// TIA Portal V16 program export: 8 tag tables, 6 data types, 67 data blocks, 106 code blocks (in call order from the OBs), 61 instance data blocks

VAR_GLOBAL   // PLC tag table "Default tag table"
   START AT %M0.0 : Bool;
   OUTPUT AT %M0.2 : Bool;
   STOP AT %M0.1 : Bool;
   MW100 AT %MW100 : Int;
END_VAR

VAR_GLOBAL   // PLC tag table "Analógicas"
   FQ301_MEDIDOR_CAUDAL AT %IW16 : Word;
   PC401_SENSOR_PRESSÃO AT %IW18 : Word;
END_VAR

VAR_GLOBAL   // PLC tag table "Estados_Componentes"
   BS001A_ON AT %I1.5 : Bool;
   BS001A_DISPARO AT %I2.0 : Bool;
   BS001B_ON AT %I2.1 : Bool;
   BS001B_DISPARO AT %I2.2 : Bool;
   XV102_ABERTA AT %I2.3 : Bool;
   XV102_FECHADA AT %I2.4 : Bool;
   XV101_ABERTA AT %I2.5 : Bool;
   MX201_ON AT %I2.6 : Bool;
   MX201_DISPARO AT %I2.7 : Bool;
   BH201_ON AT %I3.0 : Bool;
   BH201_DISPARO AT %I3.1 : Bool;
   MX301_ON AT %I3.2 : Bool;
   MX301_DISPARO AT %I3.3 : Bool;
   BM401_ON AT %I3.4 : Bool;
   BM401_DISPARO AT %I3.5 : Bool;
   BS501_ON AT %I3.6 : Bool;
   BS501_DISPARO AT %I3.7 : Bool;
   MX601_ON AT %I4.0 : Bool;
   MX601_DISPARO AT %I4.1 : Bool;
   BD601_ON AT %I4.2 : Bool;
   BD601_DISPARO AT %I4.3 : Bool;
   BD602_ON AT %I4.4 : Bool;
   BD602_DISPARO AT %I4.5 : Bool;
   MX603_ON AT %I4.6 : Bool;
   MX603_DISPARO AT %I4.7 : Bool;
   BD603_ON AT %I5.0 : Bool;
   BD603_DISPARO AT %I5.1 : Bool;
   MX604_ON AT %I5.2 : Bool;
   MX604_DISPARO AT %I5.3 : Bool;
   BD604_ON AT %I5.4 : Bool;
   BD604_DISPARO AT %I5.5 : Bool;
   MX605_ON AT %I5.6 : Bool;
   MX605_DISPARO AT %I5.7 : Bool;
   BD605_ON AT %I6.0 : Bool;
   BD605_DISPARO AT %I6.1 : Bool;
   BOT_EMERGÊNCIA AT %I6.2 : Bool;
   PH201_CONT_PH AT %I6.3 : Bool;
   PH301_CONT_PH AT %I6.4 : Bool;
   TEMPERATURA_ATINGIDA AT %I6.5 : Bool;
   RH201_CONT_REDOX AT %I6.6 : Bool;
END_VAR

VAR_GLOBAL   // PLC tag table "Falhas"
   DISPARO_DIF_3Q1_32 AT %I0.0 : Bool;
   DISPARO_DIFERENCIAL_3Q3 AT %I0.1 : Bool;
   DISPARO_DIFERENCIAL_4Q1_4Q2 AT %I0.2 : Bool;
   FALHA_24VDC AT %I0.3 : Bool;
   FALHA_220VAC AT %I0.4 : Bool;
   FALHA_24VAC AT %I0.5 : Bool;
END_VAR

VAR_GLOBAL   // PLC tag table "Níveis"
   LSH001_TK00 AT %I0.6 : Bool;
   LSL001_TK00 AT %I1.0 : Bool;
   LSH501_TK05 AT %I1.3 : Bool;
   LSL501_TK05 AT %I1.4 : Bool;
   LSH101_TK01 AT %I1.1 : Bool;
   LS201_TK02 AT %IW12 : Word;
   LS301_TK03 AT %IW14 : Word;
   LSL101_TK01 AT %I1.2 : Bool;
   LSM001_TK00 AT %I0.7 : Bool;
END_VAR

VAR_GLOBAL   // PLC tag table "Saídas"
   BS001A AT %Q0.0 : Bool;
   BS001B AT %Q0.1 : Bool;
   XV101 AT %Q3.3 : Bool;
   XV102 AT %Q3.4 : Bool;
   MX201 AT %Q0.4 : Bool;
   BH201 AT %Q0.5 : Bool;
   MX301 AT %Q0.6 : Bool;
   ALIM_BM401 AT %Q0.7 : Bool;
   LIGAR_BM401 AT %Q3.1 : Bool;
   BS501 AT %Q1.1 : Bool;
   MX601 AT %Q2.0 : Bool;
   BD601 AT %Q2.1 : Bool;
   BD602 AT %Q2.2 : Bool;
   MX603 AT %Q2.3 : Bool;
   BD603 AT %Q2.4 : Bool;
   MX604 AT %Q2.5 : Bool;
   BD604 AT %Q2.6 : Bool;
   MX605 AT %Q2.7 : Bool;
   BD605 AT %Q0.2 : Bool;
   ALARME AT %Q3.2 : Bool;
END_VAR

VAR_GLOBAL   // PLC tag table "Inputs"
   "EV1.1_ABERTA" AT %I0.0 : Bool;
   "EV1.1_FECHADA" AT %I0.1 : Bool;
   "EV2.1_ABERTA" AT %I0.2 : Bool;
   "EV2.1_FECHADA" AT %I0.3 : Bool;
   "EV3.1_ABERTA" AT %I0.4 : Bool;
   "EV3.1_FECHADA" AT %I0.5 : Bool;
   "EV4.1_ABERTA" AT %I0.6 : Bool;
   "EV4.1_FECHADA" AT %I0.7 : Bool;
   "EV5.1_ABERTA" AT %I1.0 : Bool;
   "EV5.1_FECHADA" AT %I1.1 : Bool;
   "EV1.2_ABERTA" AT %I1.2 : Bool;
   "EV1.2_FECHADA" AT %I1.3 : Bool;
   "EV2.2_ABERTA" AT %I1.4 : Bool;
   "EV2.2_FECHADA" AT %I1.5 : Bool;
   "EV3.2_ABERTA" AT %I2.0 : Bool;
   "EV3.2_FECHADA" AT %I2.1 : Bool;
   "EV4.2_ABERTA" AT %I2.2 : Bool;
   "EV4.2_FECHADA" AT %I2.3 : Bool;
   "EV5.2_ABERTA" AT %I2.4 : Bool;
   "EV5.2_FECHADA" AT %I2.5 : Bool;
   PRESSOSTATO_1 AT %IW4 : Word;
   PRESSOSTATO_2 AT %IW6 : Word;
   AVARIA_BOMBA_1 AT %I2.6 : Bool;
   AVARIA_BOMBA_2 AT %I2.7 : Bool;
   AVARIA_BOMBA_3 AT %I3.0 : Bool;
END_VAR

VAR_GLOBAL   // PLC tag table "Outputs"
   "EV1.1" AT %Q0.0 : Bool;
   "EV2.1" AT %Q0.1 : Bool;
   "EV3.1" AT %Q0.2 : Bool;
   "EV4.1" AT %Q0.3 : Bool;
   "EV5.1" AT %Q0.4 : Bool;
   "EV1.2" AT %Q0.5 : Bool;
   "EV2.2" AT %Q0.6 : Bool;
   "EV3.2" AT %Q0.7 : Bool;
   "EV4.2" AT %Q1.0 : Bool;
   "EV5.2" AT %Q1.1 : Bool;
   BOMBA_1_VAR AT %Q2.0 : Bool;
   BOMBA_2_VAR AT %Q2.1 : Bool;
   BOMBA_3_RESERVA AT %Q2.2 : Bool;
   ULTRAVIOLETA AT %Q2.3 : Bool;
END_VAR

TYPE "InverterData"
// stored: IsFailsafeCompliant false
   STRUCT
      control_word : Word;
      setpoint : Real;
      ref_quantity : Struct
         speed_p2000 : Real;
         current_p2002 : Real;
         torque_p2003 : Real;
      END_STRUCT;
      status_word : Word;
      actual_speed : Real;
      actual_current : Real;
      actual_torque : Real;
      actual_alarm : Word;
      actual_fault : Word;
      RETVAL_RD : Word;
      RETVAL_WR : Word;
   END_STRUCT;
END_TYPE

TYPE "APP"
// stored: IsFailsafeCompliant false
   STRUCT
      PID_ComponenteProporzionale : DInt;
      PID_ComponenteIntegrale : DInt;
      PID_ComponenteDerivativa : DInt;
      Tiro : Int;   // Valore di tiro richiesto: 1-100 => 1-100% Setup 1, 101-200 => 1-100% Setup 2, 0 => Azzera regolatore
      Tiro1 : Int;
      Tiro2 : Int;
      TiroPrecedente : Int;   // Valore di tiro richiesto istante (n-1)
      TiroAppoggio : Int;
      ErroreAttuale : Int;   // Errore istante (n)
      ErrorePrecedente : Int;   // Errore istante (n-1)
      PID_Kp : Int;   // Kp in uso nel PID
      PID_Ki : Int;   // Ki in uso nel PID
      PID_Kd : Int;   // Kd in uso nel PID
      SetpointTiro : Int;   // Valore di setpoint del PID
      SetpointTiroRampa : Int;   // Valore di setpoint del PID iniziale a rampa
      TransitorioInizialeFase1 : Int;   // Indica che si deve eseguire la rampa iniziale (Fase 1)
      TransitorioFase3 : Int;   // Indica che si deve eseguire la rampa da velocita' alta a media (Fase 3)
      TransitorioFase4 : Int;   // Indica che si deve eseguire la rampa da velocita' media a bassa (Fase 4)
      VelocitaRotazione : Int;   // Velocita' di rotazione richiesta
      VelocitaRotazioneFase2 : Int;   // Velocita' di rotazione richiesta durante la Fase 2
      VelocitaRotazioneAppoggio1 : Int;
      VelocitaRotazioneAppoggio2 : Int;
      Fase1OneShoot : Int;   // Indica che sono appena entrato nella fase di traansitorio di accelerazione (Fase 1)
      Fase2OneShoot : Int;   // Indica che sono appena entrato nella fase di transitorio iniziale (Fase 2)
      Fase3OneShoot : Int;   // Indica che sono appena entrato nella fase di transitorio di velocita' alta - media (Fase 3)
      Fase4OneShoot : Int;   // Indica che sono appena entrato nella fase di transitorio di velocita' media - bassa (Fase 4)
      ArrestoRepentinoOneShoot : Int;   // Indica che sono appena entrato nella fase di arresto repentino
      TiroFase1 : Int;   // Indica il tiro nella Fase 1 usato nella Fase 2
      TempIntero : Int;
      Fase : Int;
      BallerinoPrecedente : Array[0..2] of Int;   // Valore del ballerino negli istanti precedenti
      LimiteComponenteIntegrale : Int;   // Limite della componente integrale durante la transizione dalla velocita alta a media (Fase 3) e dalla media a bassa (Fase 4)
      TiroRichiesto : Int;   // Valore di tiro compreso fra 1 e 100 richiesto dalla logica di controllo
      TimerArrestoRepentino : Int;   // Timer per arresto repentino.
      TiroMinimoArrestoRepentino : Int;   // Tiro minimo durante un'arresto repentino
      VariazioneTiro : Int;   // Variazione del tiro film (ballerino)
      TimerFase2 : Int;   // Timer usato nella Fase 2 per arrestare i rulli in caso di rottura film
      TempoRotturaFilm : Int;   // Tempo rottura film in numero di scansioni (1 scansione ogni 30msec)
      TimerFase4 : Int;   // Timer per Fase 4
      TiroMinimoFase4 : Int;   // Tiro minimo durante la Fase 4 di arresto
      PID_Uscita : DInt;   // Valore di uscita del PID
      PrestiroRichiesto : DInt;   // Valore di prestiro richiesto. Valore compreso fra 0 e 500
      PrestiroAppoggio : Real;
   END_STRUCT;
END_TYPE

TYPE "DatiProgramma"
// stored: IsFailsafeCompliant false
   STRUCT
      Wrapping : Bool;   // Wrapping (0=Excluded 1=Included)
      TopLenght : Int;   // Top film lenght
      TopRelease : Int;   // Top carriage release position
      TopDown : Int;   // Top carriage downward to release top film
      Top : Int;   // Top cycle (1=Excluded 2=Before 3=Waterp-2 4=Waterp-3 5=Waterp-4)
      PressurePTime : Int;   // Time for pressure plate downward
      LifterTime : Int;   // Time for pallet lifter upward
      RevOverContrast : Int;   // Revolution over welder contrast
      RopeEndCycle : Byte;   // Rope type at end of cycle (Program)
      Spare4 : Byte;
      RopeTime : Int;   // Delay for rope unit opened
      RevOverClamp : Int;   // Revolution over clamp
      FilmForceFinalRev : Int;   // Film force on the final revolutions
      FilmPrestretchFinalRev : Int;   // Film prestretch on the final revolutions
      ArmSpeed : Int;   // Arm rotation speed (%*10)
      CarriageDown4Top : Int;   // Spool carriage downward for top cycle
      TopDownTime : Int;   // Top carriage downward for top cycle
      LapsUnderTop : Int;   // Revolutions under top film
      Spare6 : Int;   // Spare
      Spare7 : Int;   // Spare
      Spare8 : Int;   // Spare
      Spare9 : Int;   // Spare
      Spare10 : Int;   // Spare
      Spare11 : Int;   // Spare
      Spare12 : Int;   // Spare
      Overlap0_1 : Int := 0;   // Film overlap spool carriage height 0->1
      Height1 : Int := 0;   // Spool carriage height 1 (mm)
      Landmark1 : Bool := false;   // Landmark for spool carriage height 1 (0=Bottom 1=Top)
      Lifter1 : Bool := false;   // Pallet lifter for spool carriage height 1
      SpareBit1H1 : Bool := false;   // Spare bit for spool carriage height 1 (Program)
      Airblower1 : Bool := false;   // Airblower on film tail for spool carriage height 1 (0=Excluded 1=Included)
      NextStep1 : Bool := false;   // Next step for spool carriage height 1 (0=End 1=Next)
      PressureP1 : Bool := false;   // Pressure plate for spool carriage height 1 (0=Excluded 1=Included)
      SpareByte2H1 : Byte := 16#0;   // Spare byte for spool carriage height 1
      Revolution1 : Int := 0;   // Revolutions for spool carriage height 1
      RopeUnit1_1 : Byte := 16#0;   // Rope unit for spool carriage height 1 (1=Excluded 2=Inc 3=Inc during)
      RopeUnit1_2 : Byte := 16#0;   // Rope unit for spool carriage height 1 (1=Excluded 2=Inc 3=Inc during)
      FilmForce1 : Int := 0;   // Film force for spool carriage height 1
      FilmPrestretch1 : Int := 0;   // Film prestretch for spool carriage height 1
      Spare3H1 : Int := 0;   // Spare for spool carriage height 1
      Spare49 : Int := 0;   // Spare
      Spare50 : Int := 0;   // Spare
      Spare51 : Int := 0;   // Spare
      Spare52 : Int := 0;   // Spare
      Spare53 : Int := 0;   // Spare
      Overlap1_2 : Int := 0;   // Film overlap spool carriage height 1->2
      Height2 : Int := 0;   // Spool carriage height 2 (mm)
      Landmark2 : Bool := false;   // Landmark for spool carriage height 2 (0=Bottom 1=Top)
      Lifter2 : Bool := false;   // Pallet lifter for spool carriage height 2
      SpareBit1H2 : Bool := false;   // Spare bit for spool carriage height 2
      Airblower2 : Bool := false;   // Airblower on film tail for spool carriage height 2 (0=Excluded 1=Included)
      NextStep2 : Bool := false;   // Next step for spool carriage height 2 (0=End 1=Next)
      PressureP2 : Bool := false;   // Pressure plate for spool carriage height 2 (0=Excluded 1=Included)
      SpareByte2H2 : Byte := 16#0;   // Spare byte for spool carriage height 2
      Revolution2 : Int := 0;   // Revolutions for spool carriage height 2
      RopeUnit2_1 : Byte := 16#0;   // Rope unit for spool carriage height 2 (1=Excluded 2=Inc 3=Inc during)
      RopeUnit2_2 : Byte := 16#0;   // Rope unit for spool carriage height 2 (1=Excluded 2=Inc 3=Inc during)
      FilmForce2 : Int := 0;   // Film force for spool carriage height 2
      FilmPrestretch2 : Int := 0;   // Film prestretch for spool carriage height 2
      Spare3H2 : Int := 0;   // Spare for spool carriage height 2
      Spare54 : Int := 0;   // Spare
      Spare55 : Int := 0;   // Spare
      Spare56 : Int := 0;   // Spare
      Spare57 : Int := 0;   // Spare
      Spare58 : Int := 0;   // Spare
      Overlap2_3 : Int := 0;   // Film overlap spool carriage height 2->3
      Height3 : Int := 0;   // Spool carriage height 3 (mm)
      Landmark3 : Bool := false;   // Landmark for spool carriage height 3 (0=Bottom 1=Top)
      Lifter3 : Bool := false;   // Pallet lifter for spool carriage height 3
      SpareBit1H3 : Bool := false;   // Spare bit for spool carriage height 3
      Airblower3 : Bool := false;   // Airblower on film tail for spool carriage height 3 (0=Excluded 1=Included)
      NextStep3 : Bool := false;   // Next step for spool carriage height 3 (0=End 1=Next)
      PressureP3 : Bool := false;   // Pressure plate for spool carriage height 3 (0=Excluded 1=Included)
      SpareByte2H3 : Byte := 16#0;   // Spare byte for spool carriage height 3
      Revolution3 : Int := 0;   // Revolutions for spool carriage height 3
      RopeUnit3_1 : Byte := 16#0;   // Rope unit for spool carriage height 3 (1=Excluded 2=Inc 3=Inc during)
      RopeUnit3_2 : Byte := 16#0;   // Rope unit for spool carriage height 3 (1=Excluded 2=Inc 3=Inc during)
      FilmForce3 : Int := 0;   // Film force for spool carriage height 3
      FilmPrestretch3 : Int := 0;   // Film prestretch for spool carriage height 3
      Spare3H3 : Int := 0;   // Spare for spool carriage height 3
      Spare59 : Int := 0;   // Spare
      Spare60 : Int := 0;   // Spare
      Spare61 : Int := 0;   // Spare
      Spare62 : Int := 0;   // Spare
      Spare63 : Int := 0;   // Spare
      Overlap3_4 : Int := 0;   // Film overlap spool carriage height 3->4
      Height4 : Int := 0;   // Spool carriage height 4 (mm)
      Landmark4 : Bool := false;   // Landmark for spool carriage height 4 (0=Bottom 1=Top)
      Lifter4 : Bool := false;   // Pallet lifter for spool carriage height 4
      SpareBit1H4 : Bool := false;   // Spare bit for spool carriage height 4
      Airblower4 : Bool := false;   // Airblower on film tail for spool carriage height 4 (0=Excluded 1=Included)
      NextStep4 : Bool := false;   // Next step for spool carriage height 4 (0=End 1=Next)
      PressureP4 : Bool := false;   // Pressure plate for spool carriage height 4 (0=Excluded 1=Included)
      SpareByte2H4 : Byte := 16#0;   // Spare byte for spool carriage height 4
      Revolution4 : Int := 0;   // Revolutions for spool carriage height 4
      RopeUnit4_1 : Byte := 16#0;   // Rope unit for spool carriage height 4 (1=Excluded 2=Inc 3=Inc during)
      RopeUnit4_2 : Byte := 16#0;   // Rope unit for spool carriage height 4 (1=Excluded 2=Inc 3=Inc during)
      FilmForce4 : Int := 0;   // Film force for spool carriage height 4
      FilmPrestretch4 : Int := 0;   // Film prestretch for spool carriage height 4
      Spare3H4 : Int := 0;   // Spare for spool carriage height 4
      Spare64 : Int := 0;   // Spare
      Spare65 : Int := 0;   // Spare
      Spare66 : Int := 0;   // Spare
      Spare67 : Int := 0;   // Spare
      Spare68 : Int := 0;   // Spare
      Overlap4_5 : Int := 0;   // Film overlap spool carriage height 4->5
      Height5 : Int := 0;   // Spool carriage height 5 (mm)
      Landmark5 : Bool := false;   // Landmark for spool carriage height 5 (0=Bottom 1=Top)
      Lifter5 : Bool := false;   // Pallet lifter for spool carriage height 5
      SpareBit1H5 : Bool := false;   // Spare bit for spool carriage height 5
      Airblower5 : Bool := false;   // Airblower on film tail for spool carriage height 5 (0=Excluded 1=Included)
      NextStep5 : Bool := false;   // Next step for spool carriage height 5 (0=End 1=Next)
      PressureP5 : Bool := false;   // Pressure plate for spool carriage height 5 (0=Excluded 1=Included)
      SpareByte2H5 : Byte := 16#0;   // Spare byte for spool carriage height 5
      Revolution5 : Int := 0;   // Revolutions for spool carriage height 5
      RopeUnit5_1 : Byte := 16#0;   // Rope unit for spool carriage height 5 (1=Excluded 2=Inc 3=Inc during)
      RopeUnit5_2 : Byte := 16#0;   // Rope unit for spool carriage height 5 (1=Excluded 2=Inc 3=Inc during)
      FilmForce5 : Int := 0;   // Film force for spool carriage height 5
      FilmPrestretch5 : Int := 0;   // Film prestretch for spool carriage height 5
      Spare3H5 : Int := 0;   // Spare for spool carriage height 5
      Spare69 : Int := 0;   // Spare
      Spare70 : Int := 0;   // Spare
      Spare71 : Int := 0;   // Spare
      Spare72 : Int := 0;   // Spare
      Spare73 : Int := 0;   // Spare
      Overlap5_6 : Int := 0;   // Film overlap spool carriage height 5->6
      Height6 : Int := 0;   // Spool carriage height 6 (mm)
      Landmark6 : Bool := false;   // Landmark for spool carriage height 6 (0=Bottom 1=Top)
      Lifter6 : Bool := false;   // Pallet lifter for spool carriage height 6
      SpareBit1H6 : Bool := false;   // Spare bit for spool carriage height 6
      Airblower6 : Bool := false;   // Airblower on film tail for spool carriage height 6 (0=Excluded 1=Included)
      NextStep6 : Bool := false;   // Next step for spool carriage height 6 (0=End 1=Next)
      PressureP6 : Bool := false;   // Pressure plate for spool carriage height 6 (0=Excluded 1=Included)
      SpareByte2H6 : Byte := 16#0;   // Spare byte for spool carriage height 6
      Revolution6 : Int := 0;   // Revolutions for spool carriage height 6
      RopeUnit6_1 : Byte := 16#0;   // Rope unit for spool carriage height 6 (1=Excluded 2=Inc 3=Inc during)
      RopeUnit6_2 : Byte := 16#0;   // Rope unit for spool carriage height 6 (1=Excluded 2=Inc 3=Inc during)
      FilmForce6 : Int := 0;   // Film force for spool carriage height 6
      FilmPrestretch6 : Int := 0;   // Film prestretch for spool carriage height 6
      Spare3H6 : Int := 0;   // Spare for spool carriage height 6
      Spare74 : Int := 0;   // Spare
      Spare75 : Int := 0;   // Spare
      Spare76 : Int := 0;   // Spare
      Spare77 : Int := 0;   // Spare
      Spare78 : Int := 0;   // Spare
      Overlap6_7 : Int := 0;   // Film overlap spool carriage height 6->7
      Height7 : Int := 0;   // Spool carriage height 7 (mm)
      Landmark7 : Bool := false;   // Landmark for spool carriage height 7 (0=Bottom 1=Top)
      Lifter7 : Bool := false;   // Pallet lifter for spool carriage height 7
      SpareBit1H7 : Bool := false;   // Spare bit for spool carriage height 7
      Airblower7 : Bool := false;   // Airblower on film tail for spool carriage height 7 (0=Excluded 1=Included)
      NextStep7 : Bool := false;   // Next step for spool carriage height 7 (0=End 1=Next)
      PressureP7 : Bool := false;   // Pressure plate for spool carriage height 7 (0=Excluded 1=Included)
      SpareByte2H7 : Byte := 16#0;   // Spare byte for spool carriage height 7
      Revolution7 : Int := 0;   // Revolutions for spool carriage height 7
      RopeUnit7_1 : Byte := 16#0;   // Rope unit for spool carriage height 7 (1=Excluded 2=Inc 3=Inc during)
      RopeUnit7_2 : Byte := 16#0;   // Rope unit for spool carriage height 7 (1=Excluded 2=Inc 3=Inc during)
      FilmForce7 : Int := 0;   // Film force for spool carriage height 7
      FilmPrestretch7 : Int := 0;   // Film prestretch for spool carriage height 7
      Spare3H7 : Int := 0;   // Spare for spool carriage height 7
      Spare79 : Int := 0;   // Spare
      Spare80 : Int := 0;   // Spare
      Spare81 : Int := 0;   // Spare
      Spare82 : Int := 0;   // Spare
      Spare83 : Int := 0;   // Spare
      Overlap7_8 : Int := 0;   // Film overlap spool carriage height 7->8
      Height8 : Int := 0;   // Spool carriage height 8 (mm)
      Landmark8 : Bool := false;   // Landmark for spool carriage height 8 (0=Bottom 1=Top)
      Lifter8 : Bool := false;   // Pallet lifter for spool carriage height 8
      SpareBit1H8 : Bool := false;   // Spare bit for spool carriage height 8
      Airblower8 : Bool := false;   // Airblower on film tail for spool carriage height 8 (0=Excluded 1=Included)
      NextStep8 : Bool := false;   // Next step for spool carriage height 8 (0=End 1=Next)
      PressureP8 : Bool := false;   // Pressure plate for spool carriage height 8 (0=Excluded 1=Included)
      SpareByte2H8 : Byte := 16#0;   // Spare byte for spool carriage height 8
      Revolution8 : Int := 0;   // Revolutions for spool carriage height 8
      RopeUnit8_1 : Byte := 16#0;   // Rope unit for spool carriage height 8 (1=Excluded 2=Inc 3=Inc during)
      RopeUnit8_2 : Byte := 16#0;   // Rope unit for spool carriage height 8 (1=Excluded 2=Inc 3=Inc during)
      FilmForce8 : Int := 0;   // Film force for spool carriage height 8
      FilmPrestretch8 : Int := 0;   // Film prestretch for spool carriage height 8
      Spare3H8 : Int := 0;   // Spare for spool carriage height 8
      Spare84 : Int := 0;   // Spare
      Spare85 : Int := 0;   // Spare
      Spare86 : Int := 0;   // Spare
      Spare87 : Int := 0;   // Spare
      Spare88 : Int := 0;   // Spare
      Overlap8_9 : Int := 0;   // Film overlap spool carriage height 8->9
      Height9 : Int := 0;   // Spool carriage height 9 (mm)
      Landmark9 : Bool := false;   // Landmark for spool carriage height 9 (0=Bottom 1=Top)
      Lifter9 : Bool := false;   // Pallet lifter for spool carriage height 9
      SpareBit1H9 : Bool := false;   // Spare bit for spool carriage height 9
      Airblower9 : Bool := false;   // Airblower on film tail for spool carriage height 9 (0=Excluded 1=Included)
      NextStep9 : Bool := false;   // Next step for spool carriage height 9 (0=End 1=Next)
      PressureP9 : Bool := false;   // Pressure plate for spool carriage height 9 (0=Excluded 1=Included)
      SpareByte2H9 : Byte := 16#0;   // Spare byte for spool carriage height 9
      Revolution9 : Int := 0;   // Revolutions for spool carriage height 9
      RopeUnit9_1 : Byte := 16#0;   // Rope unit for spool carriage height 9 (1=Excluded 2=Inc 3=Inc during)
      RopeUnit9_2 : Byte := 16#0;   // Rope unit for spool carriage height 9 (1=Excluded 2=Inc 3=Inc during)
      FilmForce9 : Int := 0;   // Film force for spool carriage height 9
      FilmPrestretch9 : Int := 0;   // Film prestretch for spool carriage height 9
      Spare3H9 : Int := 0;   // Spare for spool carriage height 9
      Spare89 : Int := 0;   // Spare
      Spare90 : Int := 0;   // Spare
      Spare91 : Int := 0;   // Spare
      Spare92 : Int := 0;   // Spare
      Spare93 : Int := 0;   // Spare
      Overlap9_10 : Int := 0;   // Film overlap spool carriage height 9->10
      Height10 : Int := 0;   // Spool carriage height 10 (mm)
      Landmark10 : Bool := false;   // Landmark for spool carriage height 10 (0=Bottom 1=Top)
      Lifter10 : Bool := false;   // Pallet lifter for spool carriage height 10
      SpareBit1H10 : Bool := false;   // Spare bit for spool carriage height 10
      Airblower10 : Bool := false;   // Airblower on film tail for spool carriage height 10 (0=Excluded 1=Included)
      NextStep10 : Bool := false;   // Next step for spool carriage height 10 (0=End 1=Next)
      PressureP10 : Bool := false;   // Pressure plate for spool carriage height 10 (0=Excluded 1=Included)
      SpareByte2H10 : Byte := 16#0;   // Spare byte for spool carriage height 10
      Revolution10 : Int := 0;   // Revolutions for spool carriage height 10
      RopeUnit10_1 : Byte := 16#0;   // Rope unit for spool carriage height 10 (1=Excluded 2=Inc 3=Inc during)
      RopeUnit10_2 : Byte := 16#0;   // Rope unit for spool carriage height 10 (1=Excluded 2=Inc 3=Inc during)
      FilmForce10 : Int := 0;   // Film force for spool carriage height 10
      FilmPrestretch10 : Int := 0;   // Film prestretch for spool carriage height 10
      Spare3H10 : Int := 0;   // Spare for spool carriage height 10
      Spare94 : Int := 0;   // Spare
      Spare95 : Int := 0;   // Spare
      Spare96 : Int := 0;   // Spare
      Spare97 : Int := 0;   // Spare
      Spare98 : Int := 0;   // Spare
      Overlap10_11 : Int := 0;   // Film overlap spool carriage height 10->11
      Height11 : Int := 0;   // Spool carriage height 11 (mm)
      Landmark11 : Bool := false;   // Landmark for spool carriage height 11 (0=Bottom 1=Top)
      Lifter11 : Bool := false;   // Pallet lifter for spool carriage height 11
      SpareBit1H11 : Bool := false;   // Spare bit for spool carriage height 11
      Airblower11 : Bool := false;   // Airblower on film tail for spool carriage height 11 (0=Excluded 1=Included)
      NextStep11 : Bool := false;   // Next step for spool carriage height 11 (0=End 1=Next)
      PressureP11 : Bool := false;   // Pressure plate for spool carriage height 11 (0=Excluded 1=Included)
      SpareByte2H11 : Byte := 16#0;   // Spare byte for spool carriage height 11
      Revolution11 : Int := 0;   // Revolutions for spool carriage height 11
      RopeUnit11_1 : Byte := 16#0;   // Rope unit for spool carriage height 11 (1=Excluded 2=Inc 3=Inc during)
      RopeUnit11_2 : Byte := 16#0;   // Rope unit for spool carriage height 11 (1=Excluded 2=Inc 3=Inc during)
      FilmForce11 : Int := 0;   // Film force for spool carriage height 11
      FilmPrestretch11 : Int := 0;   // Film prestretch for spool carriage height 11
      Spare3H11 : Int := 0;   // Spare for spool carriage height 11
      Spare99 : Int := 0;   // Spare
      Spare100 : Int := 0;   // Spare
      Spare101 : Int := 0;   // Spare
      Spare102 : Int := 0;   // Spare
      Spare103 : Int := 0;   // Spare
      Overlap11_12 : Int := 0;   // Film overlap spool carriage height 11->12
      Height12 : Int := 0;   // Spool carriage height 12 (mm)
      Landmark12 : Bool := false;   // Landmark for spool carriage height 12 (0=Bottom 1=Top)
      Lifter12 : Bool := false;   // Pallet lifter for spool carriage height 12
      SpareBit1H12 : Bool := false;   // Spare bit for spool carriage height 12
      Airblower12 : Bool := false;   // Airblower on film tail for spool carriage height 12 (0=Excluded 1=Included)
      NextStep12 : Bool := false;   // Next step for spool carriage height 12 (0=End 1=Next)
      PressureP12 : Bool := false;   // Pressure plate for spool carriage height 12 (0=Excluded 1=Included)
      SpareByte2H12 : Byte := 16#0;   // Spare byte for spool carriage height 12
      Revolution12 : Int := 0;   // Revolutions for spool carriage height 12
      RopeUnit12_1 : Byte := 16#0;   // Rope unit for spool carriage height 12 (1=Excluded 2=Inc 3=Inc during)
      RopeUnit12_2 : Byte := 16#0;   // Rope unit for spool carriage height 12 (1=Excluded 2=Inc 3=Inc during)
      FilmForce12 : Int := 0;   // Film force for spool carriage height 12
      FilmPrestretch12 : Int := 0;   // Film prestretch for spool carriage height 12
      Spare3H12 : Int := 0;   // Spare for spool carriage height 12
      Spare104 : Int := 0;   // Spare
      Spare105 : Int := 0;   // Spare
      Spare106 : Int := 0;   // Spare
      Spare107 : Int := 0;   // Spare
      Spare108 : Int := 0;   // Spare
   END_STRUCT;
END_TYPE

TYPE "M20"
// stored: IsFailsafeCompliant false
   STRUCT
      M20_P00 : Int;   // Tipo di prestiro
      M20_P01 : Int;   // Coefficiente proporzionale per il regolatore PID
      M20_P02 : Int;   // Coefficiente integrale (Fase1 e Fase2) per il regolatore PID
      M20_P03 : Int;   // Coefficiente derivativo per il regolatore PID
      M20_P04 : Int;   // Coefficiente integrale (Fase3 e Fase4) per il regolatore PID
      M20_P05 : Int;   // Rampa di accelerazione per il tiro durante la Fase1
      M20_P06 : Int;   // Limite componente integrale nel transitorio dalla Fase2 alla Fase3
      M20_P07 : Int;   // Limite componente integrale nel transitorio dalla Fase3 alla Fase4
      M20_P08 : Int;   // Valore minimo ingresso analogico
      M20_P09 : Int;   // Valore massimo ingresso analogico
      M20_P10 : Int;   // Prestiro naturale dovuto al rapporto di riduzione
      M20_P11 : Int;   // Velocità per il jog in manuale dei rulli di prestiro
      M20_P12 : Int;   // Offset del rullo lento 10 equivale a 0
      M20_P13 : Int;   // Jog di velocità durante la partenza del braccio
      M20_P14 : Int;   // Tiro minimo durante la Fase4 di arresto e durante un arresto repentino
      M20_P15 : Int;   // Tempo (in decimi di secondo) dopo il quale i rulli si fermano per rottura film
      M20_P20 : Int;   // Velocità indicata da plc per la rotazione braccio e il carrello top
      M20_P21 : Int;   // Velocità indicata da plc per il carrello di prestiro e il trasporto di centro macchina
      M20_P22 : Int;   // Tiro indicato da plc
      M20_P23 : Int;   // Prestiro indicato da plc
      M20_P24 : Int;   // Valore di ingresso analogico AI0
      M20_P25 : Int;   // Tiro richiesto da plc compreso fra 0 e 100
   END_STRUCT;
END_TYPE

TYPE "PID"
// stored: IsFailsafeCompliant false
   STRUCT
      proporzionale : DInt;
      integrativo : DInt;
      segnale : DInt;
      maxSegnale : Int;
      minSegnale : Int;
      setPointShow : UInt;
      tiro : UInt;
      vParP : UInt;
      vParI : UInt;
      svuota : Bool;
      attiva : Bool;
      setTiro : Bool;
      "timer" : Time;
   END_STRUCT;
END_TYPE

TYPE "ProgramDataGreyBar"
// stored: IsFailsafeCompliant false
   STRUCT
      Overlap : Int;   // Film overlap
      Height : Int;   // Spool carriage height (mm)
      Landmark : Bool;   // Landmark (0=Bottom 1=Top)
      Lifter : Bool;   // Pallet lifter
      SpareBit1 : Bool;   // Spare
      Airblower : Bool;   // Airblower on film tail (0=Excluded 1=Included)
      NextStep : Bool;   // Next step (0=End 1=Next)
      PressureP : Bool;   // Pressure plate (0=Excluded 1=Included)
      SpareByte1 : Byte;   // Spare
      Revolution : Int;   // Revolutions
      RopeUnitUpper : Byte;   // Upper rope unit (1=Exc 2=Inc 3=Inc during)
      RopeUnitLower : Byte;   // Lower rope unit (1=Exc 2=Inc 3=Inc during)
      FilmForce : Int;   // Film force
      FilmPrestretch : Int;   // Film prestretch
      SpareWord1 : Int;   // Spare
      SpareWord2 : Int;   // Spare
      SpareWord3 : Int;   // Spare
      SpareWord4 : Int;   // Spare
      SpareWord5 : Int;   // Spare
      SpareWord6 : Int;   // Spare
   END_STRUCT;
END_TYPE

DATA_BLOCK "Data_block_1"   // DB1
{ S7_Optimized_Access := 'TRUE' }
VERSION : 0.1
// stored: AutoNumber true, DBAccessibleFromOPCUA true, IsOnlyStoredInLoadMemory false, IsRetainMemResEnabled false, IsWriteProtectedInAS false, MemoryReserve 100
   VAR
      DADOS : Byte;
   END_VAR
BEGIN
END_DATA_BLOCK

DATA_BLOCK "DB04_Conveyor"   // DB4
{ S7_Optimized_Access := 'FALSE' }
AUTHOR : Robopac
VERSION : 0.0
// stored: AutoNumber false, IsOnlyStoredInLoadMemory false, IsWriteProtectedInAS false
   VAR RETAIN
      dbw0 : Int := 0;
      dbw2 : Int := 0;
      dbx4_0 : Bool := TRUE;   // Pallet positioned
      dbx4_1 : Bool := FALSE;   // Deceleration for pallet positioning
      dbx4_2 : Bool := FALSE;   // Support memory for wrong pallet positioning emergency
      dbx4_3 : Bool := FALSE;   // Unload memory for outfeed conveyor
      dbx4_4 : Bool := TRUE;   // Support for end of transfer signal for pallet load/unload
      dbx4_5 : Bool := TRUE;   // Short pallet positioned
      dbx4_6 : Bool := TRUE;   // Pallet positioned for clampcutcycle
      dbx4_7 : Bool := FALSE;   // Pallet positioned from reverse
      dbb5 : Byte := 16#00;
      dbw6 : Int := 0;
      dbw8 : Int := 0;
      dbw10 : Int := 0;   // Pallet lenght measured in infeed (pulse)
      dbw12 : Int := 0;   // Pallet lenght measured in central machine (pulse)
      dbw14 : Int := 0;   // Pallet lenght measured in infeed (mm)
      dbw16 : Int := 0;   // Pallet lenght measured in central machine (mm)
      dbw18 : Int := 0;   // Half pallet lenght for selfcentering system
      dbw20 : Int := -100;   // Deceleration for pallet positioning on selfcentering system
      dbw22 : Int := 78;   // Support for conveyor movement speed
      dbw24 : Int := 0;
      dbw26 : Int := 0;
      dbw28 : Int := 0;
      dbw30 : Int := 0;
      dbw32 : Int := 0;
      dbw34 : Int := 0;
      dbd36 : DInt := 0;
      dbd40 : DInt := 0;
      dbd44 : DInt := 0;
      dbd48 : DInt := 0;
      dbd52 : DInt := 0;
      dbd56 : DInt := 0;
      dbd60 : DInt := 0;
      dbd64 : DInt := 0;
      dbd68 : DInt := 0;
      dbd72 : DInt := 0;
      dbw76 : Int := 0;
      dbb78 : Byte := 16#00;   // Rope unit for running spool carriage height (1=Excluded 2=Inc 3=Inc during
      dbb79 : Byte := 16#00;   // Rope unit for running spool carriage height (1=Excluded 2=Inc 3=Inc during
      dbd80 : DInt := 0;
      dbd84 : DInt := 0;
   END_VAR
BEGIN
END_DATA_BLOCK

DATA_BLOCK "DB09_TablePos"   // DB9
{ S7_Optimized_Access := 'FALSE' }
AUTHOR : Robopac
VERSION : 0.0
// stored: AutoNumber false, IsOnlyStoredInLoadMemory false, IsWriteProtectedInAS false
   VAR RETAIN
      dbx0_0 : Bool := FALSE;
      dbx0_1 : Bool := FALSE;
      dbx0_2 : Bool := TRUE;
      dbx0_3 : Bool := FALSE;
      dbx0_4 : Bool := FALSE;
      dbx0_5 : Bool := FALSE;
      dbx0_6 : Bool := FALSE;
      dbx0_7 : Bool := FALSE;
      dbx1_0 : Bool := FALSE;   // Table rotation axis movement forward
      dbx1_1 : Bool := FALSE;   // Table rotation axis movement backward
      dbx1_2 : Bool := FALSE;   // Table rotation axis movement inside low speed area
      dbx1_3 : Bool := FALSE;   // Table rotation axis movement low speed
      dbx1_4 : Bool := FALSE;   // Table rotation forward
      dbx1_5 : Bool := FALSE;   // Table rotation backward
      dbx1_6 : Bool := TRUE;
      dbx1_7 : Bool := FALSE;
      dbx2_0 : Bool := FALSE;
      dbx2_1 : Bool := FALSE;
      dbx2_2 : Bool := FALSE;
      dbx2_3 : Bool := FALSE;
      dbx2_4 : Bool := FALSE;
      dbx2_5 : Bool := FALSE;
      dbx2_6 : Bool := FALSE;
      dbx2_7 : Bool := FALSE;
      dbx3_0 : Bool := FALSE;   // Table rotation: Support for encoder running control
      dbx3_1 : Bool := FALSE;   // Table rotation: Support for encoder running control alarm
      dbx3_2 : Bool := FALSE;
      dbx3_3 : Bool := FALSE;
      dbx3_4 : Bool := FALSE;
      dbx3_5 : Bool := FALSE;
      dbx3_6 : Bool := FALSE;
      dbx3_7 : Bool := FALSE;
      dbx4_0 : Bool := FALSE;
      dbx4_1 : Bool := FALSE;
      dbx4_2 : Bool := FALSE;
      dbx4_3 : Bool := FALSE;
      dbx4_4 : Bool := FALSE;
      dbx4_5 : Bool := FALSE;
      dbx4_6 : Bool := FALSE;
      dbx4_7 : Bool := FALSE;
      dbx5_0 : Bool := FALSE;
      dbx5_1 : Bool := FALSE;
      dbx5_2 : Bool := FALSE;
      dbx5_3 : Bool := FALSE;
      dbw6 : Int := 5;   // Table rotation: Support for movement speed
      dbw8 : Int := 0;   // Table rotation: Support for movement deceleration
      dbw10 : Int := 5;   // Table rotation inverter: Support for speed selection
      dbw12 : Int := 10199;
      dbw14 : Int := 2340;
      dbw16 : Int := 0;
      dbw18 : Int := 0;
      dbw20 : Int := 0;
      dbw22 : Int := 0;
      dbw24 : Int := 0;
      dbw26 : Int := 0;
      dbw28 : Int := 0;
      dbd30 : DInt := -15;   // Table rotation position: Pulse
      dbw34 : Int := -8;   // Table position
      dbw36 : Int := 0;   // Table rotation position: Table maximum position
      dbw38 : Int := 0;   // Table rotation position: Deceleration position
      dbw40 : Int := 0;   // Table rotation position: Deceleration position
      dbd42 : DInt := -15;   // Support for encoder table rotation running control
      dbw46 : Int := 20;   // Support for encoder table rotation running control
      dbw48 : Int := -8;   // Table position according to offset
      dbw50 : Int := 0;
      dbw52 : Int := 0;
      dbw54 : Int := 0;
      dbw56 : Int := 0;
      dbw58 : Int := 0;
      dbw60 : Int := 0;
      dbw62 : Int := 0;
      dbw64 : Int := 0;
      dbw66 : Int := 0;
      dbw68 : Int := 0;
      dbw70 : Int := 0;
      Req1_Dest : Int := 0;   // Positioning request 1: Destination position
      Req2_Dest : Int := 0;   // Positioning request 2: Destination position
      Req3_Dest : Int := 0;   // Positioning request 3: Destination position
      Req4_Dest : Int := 0;   // Positioning request 4: Destination position
      Req1_Fwd : Bool := FALSE;   // Positioning request 1: Axis forward
      Req1_Bkw : Bool := FALSE;   // Positioning request 1: Axis backward
      Req1_Slow : Bool := FALSE;   // Positioning request 1: Axis slow speed
      Req1_Pos : Bool := FALSE;   // Positioning request 1: Axis in position
      Req2_Fwd : Bool := FALSE;   // Positioning request 2: Axis forward
      Req2_Bkw : Bool := FALSE;   // Positioning request 2: Axis backward
      Req2_Slow : Bool := FALSE;   // Positioning request 2: Axis slow speed
      Req2_Pos : Bool := FALSE;   // Positioning request 2: Axis in position
      Req3_Fwd : Bool := FALSE;   // Positioning request 3: Axis forward
      Req3_Bkw : Bool := FALSE;   // Positioning request 3: Axis backward
      Req3_Slow : Bool := FALSE;   // Positioning request 3: Axis slow speed
      Req3_Pos : Bool := FALSE;   // Positioning request 3: Axis in position
      Req4_Fwd : Bool := FALSE;   // Positioning request 4: Axis forward
      Req4_Bkw : Bool := FALSE;   // Positioning request 4: Axis backward
      Req4_Slow : Bool := FALSE;   // Positioning request 4: Axis slow speed
      Req4_Pos : Bool := FALSE;   // Positioning request 4: Axis in position
      Req5_Dest : Int := 0;   // Positioning request 4: Destination position
      Req6_Dest : Int := 0;   // Positioning request 4: Destination position
      Req7_Dest : Int := 0;   // Positioning request 4: Destination position
      Req8_Dest : Int := 0;   // Positioning request 4: Destination position
      Req5_Fwd : Bool := FALSE;   // Positioning request 5: Axis forward
      Req5_Bkw : Bool := FALSE;   // Positioning request 5: Axis backward
      Req5_Slow : Bool := FALSE;   // Positioning request 5: Axis slow speed
      Req5_Pos : Bool := FALSE;   // Positioning request 5: Axis in position
      Req6_Fwd : Bool := FALSE;   // Positioning request 6: Axis forward
      Req6_Bkw : Bool := FALSE;   // Positioning request 6: Axis backward
      Req6_Slow : Bool := FALSE;   // Positioning request 6: Axis slow speed
      Req6_Pos : Bool := FALSE;   // Positioning request 6: Axis in position
      Req7_Fwd : Bool := FALSE;   // Positioning request 7: Axis forward
      Req7_Bkw : Bool := FALSE;   // Positioning request 7: Axis backward
      Req7_Slow : Bool := FALSE;   // Positioning request 7: Axis slow speed
      Req7_Pos : Bool := FALSE;   // Positioning request 7: Axis in position
      Req8_Fwd : Bool := FALSE;   // Positioning request 8: Axis forward
      Req8_Bkw : Bool := FALSE;   // Positioning request 8: Axis backward
      Req8_Slow : Bool := FALSE;   // Positioning request 8: Axis slow speed
      Req8_Pos : Bool := FALSE;   // Positioning request 8: Axis in position
      dbw92 : Int := 0;
      dbw94 : Int := 0;
      dbw96 : Int := 0;
      dbw98 : Int := 0;
   END_VAR
BEGIN
END_DATA_BLOCK

DATA_BLOCK "DB13_TableFaseControl"   // DB13
{ S7_Optimized_Access := 'FALSE' }
VERSION : 0.1
// stored: AutoNumber false, IsOnlyStoredInLoadMemory false, IsWriteProtectedInAS false
   VAR RETAIN
      load : Bool := TRUE;
      cm : Bool := TRUE;
      unload : Bool := TRUE;
      hysteresis : Int := 100;
   END_VAR
BEGIN
END_DATA_BLOCK

DATA_BLOCK "DB18_TableSpeed"   // DB18
{ S7_Optimized_Access := 'FALSE' }
VERSION : 0.1
// stored: AutoNumber false, IsOnlyStoredInLoadMemory false, IsWriteProtectedInAS false
   VAR RETAIN
      spare0 : Int := 0;
      spare1 : Int := 0;
      spare2 : Int := 0;
      spare3 : Int := 0;
      spare4 : Int := 0;
      spare5 : Int := 0;
      spare6 : Int := 0;
      spare7 : Int := 0;
      DBD16 : Real := 0.0;   // Actual speed in degrees per second (split before use)
      DBD20 : Real := 90.0;   // Low speed in degrees per second (split before use)
      DBD24 : Real := 900.0;   // High speed in degrees per second (split before use)
      spare14 : Int := 0;
      DBW30 : Int := 0;   // Degrees to reach minimum speed from maximum speed
      spare16 : Int := 0;
      DBW34 : Int := 50;
   END_VAR
BEGIN
END_DATA_BLOCK

DATA_BLOCK "DB21_DisplayGeneralData"   // DB21
{ S7_Optimized_Access := 'FALSE' }
AUTHOR : Robopac
VERSION : 0.0
// stored: AutoNumber false, IsOnlyStoredInLoadMemory false, IsWriteProtectedInAS false
   VAR RETAIN
      dbx0_0 : Bool := TRUE;   // Welder unit included(1)/excluded (Display-General Data)
      dbx0_1 : Bool := FALSE;   // Machine included(1)/excluded (Display-General Data)
      dbx0_2 : Bool := TRUE;   // Pallet load/unload included(1)/excluded (Display-Sysdata)
      dbx0_3 : Bool := TRUE;   // Load pallet with forklift selection by display (Display-Sysdata)
      dbx0_4 : Bool := TRUE;   // Unload pallet with forklift selection by display (Display-Sysdata)
      dbx0_5 : Bool := FALSE;
      dbx0_6 : Bool := TRUE;
      dbx0_7 : Bool := FALSE;
      dbb1 : Byte := 16#00;
      dbw2 : Int := 3;   // PLC SW major release
      dbw4 : Int := 0;   // PLC SW minor release
      dbw6 : Int := 90;   // Spool carriage upward for spring clamp at begin cycle (Display-General Data)
      dbw8 : Int := 0;   // Spool carriage downward for film tail at the cycle begin (Display-General Data)
      dbw10 : Int := 2;   // Film thickness (Display-General Data)
      dbw12 : Int := 700;   // Welding time (Display-General Data)
      dbw14 : Int := 0;   // Low speed for Helix conveyor movement (%) (Display-Sysdata)
      dbw16 : Int := 0;   // High speed for Helix conveyor movement (%) (Display-Sysdata)
      dbw18 : Int := 500;   // Delay on pallet positioning (Display-General Data)
      dbw20 : Int := 10000;   // Delay for load/unload pallet simultaneously (Display-General Data)
      dbw22 : Int := 100;   // Deceleration for pallet positioning (Display-General Data)
      dbw24 : Int := 1;   // Time for pallet load with forklift
      dbw26 : Int := 0;   // Override for ring movement in manul mode (Display-General Data)
      dbw28 : Int := 100;   // TIMER CICLO FIERA (attesa tra cicli successivi)
      dbw30 : Int := 0;   // Film prestretch for film prestretch test cycle (Display-General Data)
      dbw32 : Int := 0;   // Film prestretch increase for film prestretch test (Display-General Data)
      dbw34 : Int := 0;   // Film supplied every revolution for film prestretch test (Display-General Data)
      dbw36 : Int := 0;   // Time for spool carriage upward for table cycle (Display-Sysdata)
      dbw38 : Int := 2000;   // Time for spool carriage upward for table cycle (Display-Sysdata)
      dbw40 : Int := 15000;   // Time load with forklift
      dbw42 : Int := 10000;   // Time unload with forklift
   END_VAR
BEGIN
END_DATA_BLOCK

DATA_BLOCK "DB234_Program16"   // DB234
{ S7_Optimized_Access := 'FALSE' }
AUTHOR : Robopac
VERSION : 0.0
// stored: AutoNumber false, IsOnlyStoredInLoadMemory false, IsWriteProtectedInAS false
   VAR RETAIN
      Program16 { S7_SetPoint := 'True'} : "DatiProgramma";
   END_VAR
BEGIN
   Program16.Wrapping := FALSE;
   Program16.TopLenght := 0;
   Program16.TopRelease := 0;
   Program16.TopDown := 0;
   Program16.Top := 0;
   Program16.PressurePTime := 0;
   Program16.LifterTime := 0;
   Program16.RevOverContrast := 0;
   Program16.RopeEndCycle := 16#00;
   Program16.Spare4 := 16#00;
   Program16.RopeTime := 0;
   Program16.RevOverClamp := 0;
   Program16.FilmForceFinalRev := 0;
   Program16.FilmPrestretchFinalRev := 0;
   Program16.ArmSpeed := 0;
   Program16.CarriageDown4Top := 0;
   Program16.TopDownTime := 0;
   Program16.LapsUnderTop := 0;
   Program16.Spare6 := 0;
   Program16.Spare7 := 0;
   Program16.Spare8 := 0;
   Program16.Spare9 := 0;
   Program16.Spare10 := 0;
   Program16.Spare11 := 0;
   Program16.Spare12 := 0;
   Program16.Overlap0_1 := 0;
   Program16.Height1 := 0;
   Program16.Landmark1 := FALSE;
   Program16.Lifter1 := FALSE;
   Program16.SpareBit1H1 := FALSE;
   Program16.Airblower1 := FALSE;
   Program16.NextStep1 := FALSE;
   Program16.PressureP1 := FALSE;
   Program16.SpareByte2H1 := 16#00;
   Program16.Revolution1 := 0;
   Program16.RopeUnit1_1 := 16#00;
   Program16.RopeUnit1_2 := 16#00;
   Program16.FilmForce1 := 0;
   Program16.FilmPrestretch1 := 0;
   Program16.Spare3H1 := 0;
   Program16.Spare49 := 0;
   Program16.Spare50 := 0;
   Program16.Spare51 := 0;
   Program16.Spare52 := 0;
   Program16.Spare53 := 0;
   Program16.Overlap1_2 := 0;
   Program16.Height2 := 0;
   Program16.Landmark2 := FALSE;
   Program16.Lifter2 := FALSE;
   Program16.SpareBit1H2 := FALSE;
   Program16.Airblower2 := FALSE;
   Program16.NextStep2 := FALSE;
   Program16.PressureP2 := FALSE;
   Program16.SpareByte2H2 := 16#00;
   Program16.Revolution2 := 0;
   Program16.RopeUnit2_1 := 16#00;
   Program16.RopeUnit2_2 := 16#00;
   Program16.FilmForce2 := 0;
   Program16.FilmPrestretch2 := 0;
   Program16.Spare3H2 := 0;
   Program16.Spare54 := 0;
   Program16.Spare55 := 0;
   Program16.Spare56 := 0;
   Program16.Spare57 := 0;
   Program16.Spare58 := 0;
   Program16.Overlap2_3 := 0;
   Program16.Height3 := 0;
   Program16.Landmark3 := FALSE;
   Program16.Lifter3 := FALSE;
   Program16.SpareBit1H3 := FALSE;
   Program16.Airblower3 := FALSE;
   Program16.NextStep3 := FALSE;
   Program16.PressureP3 := FALSE;
   Program16.SpareByte2H3 := 16#00;
   Program16.Revolution3 := 0;
   Program16.RopeUnit3_1 := 16#00;
   Program16.RopeUnit3_2 := 16#00;
   Program16.FilmForce3 := 0;
   Program16.FilmPrestretch3 := 0;
   Program16.Spare3H3 := 0;
   Program16.Spare59 := 0;
   Program16.Spare60 := 0;
   Program16.Spare61 := 0;
   Program16.Spare62 := 0;
   Program16.Spare63 := 0;
   Program16.Overlap3_4 := 0;
   Program16.Height4 := 0;
   Program16.Landmark4 := FALSE;
   Program16.Lifter4 := FALSE;
   Program16.SpareBit1H4 := FALSE;
   Program16.Airblower4 := FALSE;
   Program16.NextStep4 := FALSE;
   Program16.PressureP4 := FALSE;
   Program16.SpareByte2H4 := 16#00;
   Program16.Revolution4 := 0;
   Program16.RopeUnit4_1 := 16#00;
   Program16.RopeUnit4_2 := 16#00;
   Program16.FilmForce4 := 0;
   Program16.FilmPrestretch4 := 0;
   Program16.Spare3H4 := 0;
   Program16.Spare64 := 0;
   Program16.Spare65 := 0;
   Program16.Spare66 := 0;
   Program16.Spare67 := 0;
   Program16.Spare68 := 0;
   Program16.Overlap4_5 := 0;
   Program16.Height5 := 0;
   Program16.Landmark5 := FALSE;
   Program16.Lifter5 := FALSE;
   Program16.SpareBit1H5 := FALSE;
   Program16.Airblower5 := FALSE;
   Program16.NextStep5 := FALSE;
   Program16.PressureP5 := FALSE;
   Program16.SpareByte2H5 := 16#00;
   Program16.Revolution5 := 0;
   Program16.RopeUnit5_1 := 16#00;
   Program16.RopeUnit5_2 := 16#00;
   Program16.FilmForce5 := 0;
   Program16.FilmPrestretch5 := 0;
   Program16.Spare3H5 := 0;
   Program16.Spare69 := 0;
   Program16.Spare70 := 0;
   Program16.Spare71 := 0;
   Program16.Spare72 := 0;
   Program16.Spare73 := 0;
   Program16.Overlap5_6 := 0;
   Program16.Height6 := 0;
   Program16.Landmark6 := FALSE;
   Program16.Lifter6 := FALSE;
   Program16.SpareBit1H6 := FALSE;
   Program16.Airblower6 := FALSE;
   Program16.NextStep6 := FALSE;
   Program16.PressureP6 := FALSE;
   Program16.SpareByte2H6 := 16#00;
   Program16.Revolution6 := 0;
   Program16.RopeUnit6_1 := 16#00;
   Program16.RopeUnit6_2 := 16#00;
   Program16.FilmForce6 := 0;
   Program16.FilmPrestretch6 := 0;
   Program16.Spare3H6 := 0;
   Program16.Spare74 := 0;
   Program16.Spare75 := 0;
   Program16.Spare76 := 0;
   Program16.Spare77 := 0;
   Program16.Spare78 := 0;
   Program16.Overlap6_7 := 0;
   Program16.Height7 := 0;
   Program16.Landmark7 := FALSE;
   Program16.Lifter7 := FALSE;
   Program16.SpareBit1H7 := FALSE;
   Program16.Airblower7 := FALSE;
   Program16.NextStep7 := FALSE;
   Program16.PressureP7 := FALSE;
   Program16.SpareByte2H7 := 16#00;
   Program16.Revolution7 := 0;
   Program16.RopeUnit7_1 := 16#00;
   Program16.RopeUnit7_2 := 16#00;
   Program16.FilmForce7 := 0;
   Program16.FilmPrestretch7 := 0;
   Program16.Spare3H7 := 0;
   Program16.Spare79 := 0;
   Program16.Spare80 := 0;
   Program16.Spare81 := 0;
   Program16.Spare82 := 0;
   Program16.Spare83 := 0;
   Program16.Overlap7_8 := 0;
   Program16.Height8 := 0;
   Program16.Landmark8 := FALSE;
   Program16.Lifter8 := FALSE;
   Program16.SpareBit1H8 := FALSE;
   Program16.Airblower8 := FALSE;
   Program16.NextStep8 := FALSE;
   Program16.PressureP8 := FALSE;
   Program16.SpareByte2H8 := 16#00;
   Program16.Revolution8 := 0;
   Program16.RopeUnit8_1 := 16#00;
   Program16.RopeUnit8_2 := 16#00;
   Program16.FilmForce8 := 0;
   Program16.FilmPrestretch8 := 0;
   Program16.Spare3H8 := 0;
   Program16.Spare84 := 0;
   Program16.Spare85 := 0;
   Program16.Spare86 := 0;
   Program16.Spare87 := 0;
   Program16.Spare88 := 0;
   Program16.Overlap8_9 := 0;
   Program16.Height9 := 0;
   Program16.Landmark9 := FALSE;
   Program16.Lifter9 := FALSE;
   Program16.SpareBit1H9 := FALSE;
   Program16.Airblower9 := FALSE;
   Program16.NextStep9 := FALSE;
   Program16.PressureP9 := FALSE;
   Program16.SpareByte2H9 := 16#00;
   Program16.Revolution9 := 0;
   Program16.RopeUnit9_1 := 16#00;
   Program16.RopeUnit9_2 := 16#00;
   Program16.FilmForce9 := 0;
   Program16.FilmPrestretch9 := 0;
   Program16.Spare3H9 := 0;
   Program16.Spare89 := 0;
   Program16.Spare90 := 0;
   Program16.Spare91 := 0;
   Program16.Spare92 := 0;
   Program16.Spare93 := 0;
   Program16.Overlap9_10 := 0;
   Program16.Height10 := 0;
   Program16.Landmark10 := FALSE;
   Program16.Lifter10 := FALSE;
   Program16.SpareBit1H10 := FALSE;
   Program16.Airblower10 := FALSE;
   Program16.NextStep10 := FALSE;
   Program16.PressureP10 := FALSE;
   Program16.SpareByte2H10 := 16#00;
   Program16.Revolution10 := 0;
   Program16.RopeUnit10_1 := 16#00;
   Program16.RopeUnit10_2 := 16#00;
   Program16.FilmForce10 := 0;
   Program16.FilmPrestretch10 := 0;
   Program16.Spare3H10 := 0;
   Program16.Spare94 := 0;
   Program16.Spare95 := 0;
   Program16.Spare96 := 0;
   Program16.Spare97 := 0;
   Program16.Spare98 := 0;
   Program16.Overlap10_11 := 0;
   Program16.Height11 := 0;
   Program16.Landmark11 := FALSE;
   Program16.Lifter11 := FALSE;
   Program16.SpareBit1H11 := FALSE;
   Program16.Airblower11 := FALSE;
   Program16.NextStep11 := FALSE;
   Program16.PressureP11 := FALSE;
   Program16.SpareByte2H11 := 16#00;
   Program16.Revolution11 := 0;
   Program16.RopeUnit11_1 := 16#00;
   Program16.RopeUnit11_2 := 16#00;
   Program16.FilmForce11 := 0;
   Program16.FilmPrestretch11 := 0;
   Program16.Spare3H11 := 0;
   Program16.Spare99 := 0;
   Program16.Spare100 := 0;
   Program16.Spare101 := 0;
   Program16.Spare102 := 0;
   Program16.Spare103 := 0;
   Program16.Overlap11_12 := 0;
   Program16.Height12 := 0;
   Program16.Landmark12 := FALSE;
   Program16.Lifter12 := FALSE;
   Program16.SpareBit1H12 := FALSE;
   Program16.Airblower12 := FALSE;
   Program16.NextStep12 := FALSE;
   Program16.PressureP12 := FALSE;
   Program16.SpareByte2H12 := 16#00;
   Program16.Revolution12 := 0;
   Program16.RopeUnit12_1 := 16#00;
   Program16.RopeUnit12_2 := 16#00;
   Program16.FilmForce12 := 0;
   Program16.FilmPrestretch12 := 0;
   Program16.Spare3H12 := 0;
   Program16.Spare104 := 0;
   Program16.Spare105 := 0;
   Program16.Spare106 := 0;
   Program16.Spare107 := 0;
   Program16.Spare108 := 0;
END_DATA_BLOCK

DATA_BLOCK "DB236_Program14"   // DB236
{ S7_Optimized_Access := 'FALSE' }
AUTHOR : Robopac
VERSION : 0.0
// stored: AutoNumber false, IsOnlyStoredInLoadMemory false, IsWriteProtectedInAS false
   VAR RETAIN
      Program14 { S7_SetPoint := 'True'} : "DatiProgramma";
   END_VAR
BEGIN
   Program14.Wrapping := TRUE;
   Program14.TopLenght := 500;
   Program14.TopRelease := 0;
   Program14.TopDown := 0;
   Program14.Top := 4;
   Program14.PressurePTime := 0;
   Program14.LifterTime := 0;
   Program14.RevOverContrast := 1;
   Program14.RopeEndCycle := 16#02;
   Program14.Spare4 := 16#01;
   Program14.RopeTime := 1500;
   Program14.RevOverClamp := 1;
   Program14.FilmForceFinalRev := 10;
   Program14.FilmPrestretchFinalRev := 100;
   Program14.ArmSpeed := 100;
   Program14.CarriageDown4Top := 500;
   Program14.TopDownTime := 1500;
   Program14.LapsUnderTop := 0;
   Program14.Spare6 := 0;
   Program14.Spare7 := 0;
   Program14.Spare8 := 0;
   Program14.Spare9 := 0;
   Program14.Spare10 := 0;
   Program14.Spare11 := 0;
   Program14.Spare12 := 0;
   Program14.Overlap0_1 := 0;
   Program14.Height1 := 130;
   Program14.Landmark1 := FALSE;
   Program14.Lifter1 := FALSE;
   Program14.SpareBit1H1 := FALSE;
   Program14.Airblower1 := TRUE;
   Program14.NextStep1 := TRUE;
   Program14.PressureP1 := TRUE;
   Program14.SpareByte2H1 := 16#00;
   Program14.Revolution1 := 1;
   Program14.RopeUnit1_1 := 16#01;
   Program14.RopeUnit1_2 := 16#01;
   Program14.FilmForce1 := 5;
   Program14.FilmPrestretch1 := 200;
   Program14.Spare3H1 := 0;
   Program14.Spare49 := 0;
   Program14.Spare50 := 0;
   Program14.Spare51 := 0;
   Program14.Spare52 := 0;
   Program14.Spare53 := 0;
   Program14.Overlap1_2 := 0;
   Program14.Height2 := 50;
   Program14.Landmark2 := FALSE;
   Program14.Lifter2 := FALSE;
   Program14.SpareBit1H2 := FALSE;
   Program14.Airblower2 := TRUE;
   Program14.NextStep2 := TRUE;
   Program14.PressureP2 := TRUE;
   Program14.SpareByte2H2 := 16#00;
   Program14.Revolution2 := 1;
   Program14.RopeUnit2_1 := 16#01;
   Program14.RopeUnit2_2 := 16#01;
   Program14.FilmForce2 := 20;
   Program14.FilmPrestretch2 := 200;
   Program14.Spare3H2 := 0;
   Program14.Spare54 := 0;
   Program14.Spare55 := 0;
   Program14.Spare56 := 0;
   Program14.Spare57 := 0;
   Program14.Spare58 := 0;
   Program14.Overlap2_3 := 100;
   Program14.Height3 := -50;
   Program14.Landmark3 := TRUE;
   Program14.Lifter3 := FALSE;
   Program14.SpareBit1H3 := FALSE;
   Program14.Airblower3 := TRUE;
   Program14.NextStep3 := TRUE;
   Program14.PressureP3 := TRUE;
   Program14.SpareByte2H3 := 16#00;
   Program14.Revolution3 := 2;
   Program14.RopeUnit3_1 := 16#01;
   Program14.RopeUnit3_2 := 16#01;
   Program14.FilmForce3 := 30;
   Program14.FilmPrestretch3 := 200;
   Program14.Spare3H3 := 0;
   Program14.Spare59 := 0;
   Program14.Spare60 := 0;
   Program14.Spare61 := 380;
   Program14.Spare62 := 2800;
   Program14.Spare63 := 0;
   Program14.Overlap3_4 := 100;
   Program14.Height4 := 100;
   Program14.Landmark4 := FALSE;
   Program14.Lifter4 := FALSE;
   Program14.SpareBit1H4 := FALSE;
   Program14.Airblower4 := TRUE;
   Program14.NextStep4 := TRUE;
   Program14.PressureP4 := TRUE;
   Program14.SpareByte2H4 := 16#00;
   Program14.Revolution4 := 3;
   Program14.RopeUnit4_1 := 16#02;
   Program14.RopeUnit4_2 := 16#02;
   Program14.FilmForce4 := 30;
   Program14.FilmPrestretch4 := 200;
   Program14.Spare3H4 := 0;
   Program14.Spare64 := 0;
   Program14.Spare65 := 0;
   Program14.Spare66 := 0;
   Program14.Spare67 := 0;
   Program14.Spare68 := 0;
   Program14.Overlap4_5 := 0;
   Program14.Height5 := 50;
   Program14.Landmark5 := FALSE;
   Program14.Lifter5 := FALSE;
   Program14.SpareBit1H5 := FALSE;
   Program14.Airblower5 := TRUE;
   Program14.NextStep5 := FALSE;
   Program14.PressureP5 := FALSE;
   Program14.SpareByte2H5 := 16#00;
   Program14.Revolution5 := 1;
   Program14.RopeUnit5_1 := 16#01;
   Program14.RopeUnit5_2 := 16#01;
   Program14.FilmForce5 := 30;
   Program14.FilmPrestretch5 := 200;
   Program14.Spare3H5 := 0;
   Program14.Spare69 := 0;
   Program14.Spare70 := 0;
   Program14.Spare71 := 0;
   Program14.Spare72 := 0;
   Program14.Spare73 := 0;
   Program14.Overlap5_6 := 100;
   Program14.Height6 := 50;
   Program14.Landmark6 := FALSE;
   Program14.Lifter6 := FALSE;
   Program14.SpareBit1H6 := FALSE;
   Program14.Airblower6 := TRUE;
   Program14.NextStep6 := FALSE;
   Program14.PressureP6 := FALSE;
   Program14.SpareByte2H6 := 16#00;
   Program14.Revolution6 := 2;
   Program14.RopeUnit6_1 := 16#02;
   Program14.RopeUnit6_2 := 16#01;
   Program14.FilmForce6 := 20;
   Program14.FilmPrestretch6 := 200;
   Program14.Spare3H6 := 0;
   Program14.Spare74 := 0;
   Program14.Spare75 := 0;
   Program14.Spare76 := 0;
   Program14.Spare77 := 0;
   Program14.Spare78 := 0;
   Program14.Overlap6_7 := 0;
   Program14.Height7 := 0;
   Program14.Landmark7 := FALSE;
   Program14.Lifter7 := FALSE;
   Program14.SpareBit1H7 := FALSE;
   Program14.Airblower7 := FALSE;
   Program14.NextStep7 := TRUE;
   Program14.PressureP7 := FALSE;
   Program14.SpareByte2H7 := 16#00;
   Program14.Revolution7 := 1;
   Program14.RopeUnit7_1 := 16#01;
   Program14.RopeUnit7_2 := 16#01;
   Program14.FilmForce7 := 0;
   Program14.FilmPrestretch7 := 100;
   Program14.Spare3H7 := 0;
   Program14.Spare79 := 0;
   Program14.Spare80 := 0;
   Program14.Spare81 := 0;
   Program14.Spare82 := 0;
   Program14.Spare83 := 0;
   Program14.Overlap7_8 := 0;
   Program14.Height8 := 0;
   Program14.Landmark8 := FALSE;
   Program14.Lifter8 := FALSE;
   Program14.SpareBit1H8 := FALSE;
   Program14.Airblower8 := FALSE;
   Program14.NextStep8 := TRUE;
   Program14.PressureP8 := FALSE;
   Program14.SpareByte2H8 := 16#00;
   Program14.Revolution8 := 1;
   Program14.RopeUnit8_1 := 16#01;
   Program14.RopeUnit8_2 := 16#01;
   Program14.FilmForce8 := 0;
   Program14.FilmPrestretch8 := 100;
   Program14.Spare3H8 := 0;
   Program14.Spare84 := 0;
   Program14.Spare85 := 0;
   Program14.Spare86 := 0;
   Program14.Spare87 := 0;
   Program14.Spare88 := 0;
   Program14.Overlap8_9 := 0;
   Program14.Height9 := 0;
   Program14.Landmark9 := FALSE;
   Program14.Lifter9 := FALSE;
   Program14.SpareBit1H9 := FALSE;
   Program14.Airblower9 := FALSE;
   Program14.NextStep9 := TRUE;
   Program14.PressureP9 := FALSE;
   Program14.SpareByte2H9 := 16#00;
   Program14.Revolution9 := 1;
   Program14.RopeUnit9_1 := 16#01;
   Program14.RopeUnit9_2 := 16#01;
   Program14.FilmForce9 := 0;
   Program14.FilmPrestretch9 := 100;
   Program14.Spare3H9 := 0;
   Program14.Spare89 := 0;
   Program14.Spare90 := 0;
   Program14.Spare91 := 0;
   Program14.Spare92 := 0;
   Program14.Spare93 := 0;
   Program14.Overlap9_10 := 0;
   Program14.Height10 := 0;
   Program14.Landmark10 := FALSE;
   Program14.Lifter10 := FALSE;
   Program14.SpareBit1H10 := FALSE;
   Program14.Airblower10 := FALSE;
   Program14.NextStep10 := FALSE;
   Program14.PressureP10 := FALSE;
   Program14.SpareByte2H10 := 16#00;
   Program14.Revolution10 := 1;
   Program14.RopeUnit10_1 := 16#01;
   Program14.RopeUnit10_2 := 16#01;
   Program14.FilmForce10 := 0;
   Program14.FilmPrestretch10 := 100;
   Program14.Spare3H10 := 0;
   Program14.Spare94 := 0;
   Program14.Spare95 := 0;
   Program14.Spare96 := 0;
   Program14.Spare97 := 0;
   Program14.Spare98 := 0;
   Program14.Overlap10_11 := 0;
   Program14.Height11 := 0;
   Program14.Landmark11 := FALSE;
   Program14.Lifter11 := FALSE;
   Program14.SpareBit1H11 := FALSE;
   Program14.Airblower11 := FALSE;
   Program14.NextStep11 := TRUE;
   Program14.PressureP11 := FALSE;
   Program14.SpareByte2H11 := 16#00;
   Program14.Revolution11 := 1;
   Program14.RopeUnit11_1 := 16#01;
   Program14.RopeUnit11_2 := 16#01;
   Program14.FilmForce11 := 0;
   Program14.FilmPrestretch11 := 100;
   Program14.Spare3H11 := 0;
   Program14.Spare99 := 0;
   Program14.Spare100 := 0;
   Program14.Spare101 := 0;
   Program14.Spare102 := 0;
   Program14.Spare103 := 0;
   Program14.Overlap11_12 := 0;
   Program14.Height12 := 0;
   Program14.Landmark12 := FALSE;
   Program14.Lifter12 := FALSE;
   Program14.SpareBit1H12 := FALSE;
   Program14.Airblower12 := FALSE;
   Program14.NextStep12 := FALSE;
   Program14.PressureP12 := FALSE;
   Program14.SpareByte2H12 := 16#00;
   Program14.Revolution12 := 1;
   Program14.RopeUnit12_1 := 16#01;
   Program14.RopeUnit12_2 := 16#01;
   Program14.FilmForce12 := 0;
   Program14.FilmPrestretch12 := 100;
   Program14.Spare3H12 := 0;
   Program14.Spare104 := 0;
   Program14.Spare105 := 0;
   Program14.Spare106 := 0;
   Program14.Spare107 := 0;
   Program14.Spare108 := 0;
END_DATA_BLOCK

DATA_BLOCK "DB237_Program13"   // DB237
{ S7_Optimized_Access := 'FALSE' }
AUTHOR : Robopac
VERSION : 0.0
// stored: AutoNumber false, IsOnlyStoredInLoadMemory false, IsWriteProtectedInAS false
   VAR RETAIN
      Program13 { S7_SetPoint := 'True'} : "DatiProgramma";
   END_VAR
BEGIN
   Program13.Wrapping := TRUE;
   Program13.TopLenght := 500;
   Program13.TopRelease := 0;
   Program13.TopDown := 0;
   Program13.Top := 4;
   Program13.PressurePTime := 0;
   Program13.LifterTime := 0;
   Program13.RevOverContrast := 1;
   Program13.RopeEndCycle := 16#02;
   Program13.Spare4 := 16#01;
   Program13.RopeTime := 1500;
   Program13.RevOverClamp := 1;
   Program13.FilmForceFinalRev := 10;
   Program13.FilmPrestretchFinalRev := 100;
   Program13.ArmSpeed := 100;
   Program13.CarriageDown4Top := 500;
   Program13.TopDownTime := 1500;
   Program13.LapsUnderTop := 0;
   Program13.Spare6 := 0;
   Program13.Spare7 := 0;
   Program13.Spare8 := 0;
   Program13.Spare9 := 0;
   Program13.Spare10 := 0;
   Program13.Spare11 := 0;
   Program13.Spare12 := 0;
   Program13.Overlap0_1 := 0;
   Program13.Height1 := 130;
   Program13.Landmark1 := FALSE;
   Program13.Lifter1 := FALSE;
   Program13.SpareBit1H1 := FALSE;
   Program13.Airblower1 := TRUE;
   Program13.NextStep1 := TRUE;
   Program13.PressureP1 := TRUE;
   Program13.SpareByte2H1 := 16#00;
   Program13.Revolution1 := 1;
   Program13.RopeUnit1_1 := 16#01;
   Program13.RopeUnit1_2 := 16#01;
   Program13.FilmForce1 := 5;
   Program13.FilmPrestretch1 := 200;
   Program13.Spare3H1 := 0;
   Program13.Spare49 := 0;
   Program13.Spare50 := 0;
   Program13.Spare51 := 0;
   Program13.Spare52 := 0;
   Program13.Spare53 := 0;
   Program13.Overlap1_2 := 0;
   Program13.Height2 := 50;
   Program13.Landmark2 := FALSE;
   Program13.Lifter2 := FALSE;
   Program13.SpareBit1H2 := FALSE;
   Program13.Airblower2 := TRUE;
   Program13.NextStep2 := TRUE;
   Program13.PressureP2 := TRUE;
   Program13.SpareByte2H2 := 16#00;
   Program13.Revolution2 := 1;
   Program13.RopeUnit2_1 := 16#01;
   Program13.RopeUnit2_2 := 16#01;
   Program13.FilmForce2 := 20;
   Program13.FilmPrestretch2 := 200;
   Program13.Spare3H2 := 0;
   Program13.Spare54 := 0;
   Program13.Spare55 := 0;
   Program13.Spare56 := 0;
   Program13.Spare57 := 0;
   Program13.Spare58 := 0;
   Program13.Overlap2_3 := 100;
   Program13.Height3 := -50;
   Program13.Landmark3 := TRUE;
   Program13.Lifter3 := FALSE;
   Program13.SpareBit1H3 := FALSE;
   Program13.Airblower3 := TRUE;
   Program13.NextStep3 := TRUE;
   Program13.PressureP3 := TRUE;
   Program13.SpareByte2H3 := 16#00;
   Program13.Revolution3 := 2;
   Program13.RopeUnit3_1 := 16#01;
   Program13.RopeUnit3_2 := 16#01;
   Program13.FilmForce3 := 30;
   Program13.FilmPrestretch3 := 200;
   Program13.Spare3H3 := 0;
   Program13.Spare59 := 0;
   Program13.Spare60 := 0;
   Program13.Spare61 := 380;
   Program13.Spare62 := 2800;
   Program13.Spare63 := 0;
   Program13.Overlap3_4 := 100;
   Program13.Height4 := 100;
   Program13.Landmark4 := FALSE;
   Program13.Lifter4 := FALSE;
   Program13.SpareBit1H4 := FALSE;
   Program13.Airblower4 := TRUE;
   Program13.NextStep4 := TRUE;
   Program13.PressureP4 := TRUE;
   Program13.SpareByte2H4 := 16#00;
   Program13.Revolution4 := 3;
   Program13.RopeUnit4_1 := 16#02;
   Program13.RopeUnit4_2 := 16#02;
   Program13.FilmForce4 := 30;
   Program13.FilmPrestretch4 := 200;
   Program13.Spare3H4 := 0;
   Program13.Spare64 := 0;
   Program13.Spare65 := 0;
   Program13.Spare66 := 0;
   Program13.Spare67 := 0;
   Program13.Spare68 := 0;
   Program13.Overlap4_5 := 0;
   Program13.Height5 := 50;
   Program13.Landmark5 := FALSE;
   Program13.Lifter5 := FALSE;
   Program13.SpareBit1H5 := FALSE;
   Program13.Airblower5 := TRUE;
   Program13.NextStep5 := FALSE;
   Program13.PressureP5 := FALSE;
   Program13.SpareByte2H5 := 16#00;
   Program13.Revolution5 := 1;
   Program13.RopeUnit5_1 := 16#01;
   Program13.RopeUnit5_2 := 16#01;
   Program13.FilmForce5 := 30;
   Program13.FilmPrestretch5 := 200;
   Program13.Spare3H5 := 0;
   Program13.Spare69 := 0;
   Program13.Spare70 := 0;
   Program13.Spare71 := 0;
   Program13.Spare72 := 0;
   Program13.Spare73 := 0;
   Program13.Overlap5_6 := 100;
   Program13.Height6 := 50;
   Program13.Landmark6 := FALSE;
   Program13.Lifter6 := FALSE;
   Program13.SpareBit1H6 := FALSE;
   Program13.Airblower6 := TRUE;
   Program13.NextStep6 := FALSE;
   Program13.PressureP6 := FALSE;
   Program13.SpareByte2H6 := 16#00;
   Program13.Revolution6 := 2;
   Program13.RopeUnit6_1 := 16#02;
   Program13.RopeUnit6_2 := 16#01;
   Program13.FilmForce6 := 20;
   Program13.FilmPrestretch6 := 200;
   Program13.Spare3H6 := 0;
   Program13.Spare74 := 0;
   Program13.Spare75 := 0;
   Program13.Spare76 := 0;
   Program13.Spare77 := 0;
   Program13.Spare78 := 0;
   Program13.Overlap6_7 := 0;
   Program13.Height7 := 0;
   Program13.Landmark7 := FALSE;
   Program13.Lifter7 := FALSE;
   Program13.SpareBit1H7 := FALSE;
   Program13.Airblower7 := FALSE;
   Program13.NextStep7 := TRUE;
   Program13.PressureP7 := FALSE;
   Program13.SpareByte2H7 := 16#00;
   Program13.Revolution7 := 1;
   Program13.RopeUnit7_1 := 16#01;
   Program13.RopeUnit7_2 := 16#01;
   Program13.FilmForce7 := 0;
   Program13.FilmPrestretch7 := 100;
   Program13.Spare3H7 := 0;
   Program13.Spare79 := 0;
   Program13.Spare80 := 0;
   Program13.Spare81 := 0;
   Program13.Spare82 := 0;
   Program13.Spare83 := 0;
   Program13.Overlap7_8 := 0;
   Program13.Height8 := 0;
   Program13.Landmark8 := FALSE;
   Program13.Lifter8 := FALSE;
   Program13.SpareBit1H8 := FALSE;
   Program13.Airblower8 := FALSE;
   Program13.NextStep8 := TRUE;
   Program13.PressureP8 := FALSE;
   Program13.SpareByte2H8 := 16#00;
   Program13.Revolution8 := 1;
   Program13.RopeUnit8_1 := 16#01;
   Program13.RopeUnit8_2 := 16#01;
   Program13.FilmForce8 := 0;
   Program13.FilmPrestretch8 := 100;
   Program13.Spare3H8 := 0;
   Program13.Spare84 := 0;
   Program13.Spare85 := 0;
   Program13.Spare86 := 0;
   Program13.Spare87 := 0;
   Program13.Spare88 := 0;
   Program13.Overlap8_9 := 0;
   Program13.Height9 := 0;
   Program13.Landmark9 := FALSE;
   Program13.Lifter9 := FALSE;
   Program13.SpareBit1H9 := FALSE;
   Program13.Airblower9 := FALSE;
   Program13.NextStep9 := TRUE;
   Program13.PressureP9 := FALSE;
   Program13.SpareByte2H9 := 16#00;
   Program13.Revolution9 := 1;
   Program13.RopeUnit9_1 := 16#01;
   Program13.RopeUnit9_2 := 16#01;
   Program13.FilmForce9 := 0;
   Program13.FilmPrestretch9 := 100;
   Program13.Spare3H9 := 0;
   Program13.Spare89 := 0;
   Program13.Spare90 := 0;
   Program13.Spare91 := 0;
   Program13.Spare92 := 0;
   Program13.Spare93 := 0;
   Program13.Overlap9_10 := 0;
   Program13.Height10 := 0;
   Program13.Landmark10 := FALSE;
   Program13.Lifter10 := FALSE;
   Program13.SpareBit1H10 := FALSE;
   Program13.Airblower10 := FALSE;
   Program13.NextStep10 := FALSE;
   Program13.PressureP10 := FALSE;
   Program13.SpareByte2H10 := 16#00;
   Program13.Revolution10 := 1;
   Program13.RopeUnit10_1 := 16#01;
   Program13.RopeUnit10_2 := 16#01;
   Program13.FilmForce10 := 0;
   Program13.FilmPrestretch10 := 100;
   Program13.Spare3H10 := 0;
   Program13.Spare94 := 0;
   Program13.Spare95 := 0;
   Program13.Spare96 := 0;
   Program13.Spare97 := 0;
   Program13.Spare98 := 0;
   Program13.Overlap10_11 := 0;
   Program13.Height11 := 0;
   Program13.Landmark11 := FALSE;
   Program13.Lifter11 := FALSE;
   Program13.SpareBit1H11 := FALSE;
   Program13.Airblower11 := FALSE;
   Program13.NextStep11 := TRUE;
   Program13.PressureP11 := FALSE;
   Program13.SpareByte2H11 := 16#00;
   Program13.Revolution11 := 1;
   Program13.RopeUnit11_1 := 16#01;
   Program13.RopeUnit11_2 := 16#01;
   Program13.FilmForce11 := 0;
   Program13.FilmPrestretch11 := 100;
   Program13.Spare3H11 := 0;
   Program13.Spare99 := 0;
   Program13.Spare100 := 0;
   Program13.Spare101 := 0;
   Program13.Spare102 := 0;
   Program13.Spare103 := 0;
   Program13.Overlap11_12 := 0;
   Program13.Height12 := 0;
   Program13.Landmark12 := FALSE;
   Program13.Lifter12 := FALSE;
   Program13.SpareBit1H12 := FALSE;
   Program13.Airblower12 := FALSE;
   Program13.NextStep12 := FALSE;
   Program13.PressureP12 := FALSE;
   Program13.SpareByte2H12 := 16#00;
   Program13.Revolution12 := 1;
   Program13.RopeUnit12_1 := 16#01;
   Program13.RopeUnit12_2 := 16#01;
   Program13.FilmForce12 := 0;
   Program13.FilmPrestretch12 := 100;
   Program13.Spare3H12 := 0;
   Program13.Spare104 := 0;
   Program13.Spare105 := 0;
   Program13.Spare106 := 0;
   Program13.Spare107 := 0;
   Program13.Spare108 := 0;
END_DATA_BLOCK

DATA_BLOCK "DB238_Program12"   // DB238
{ S7_Optimized_Access := 'FALSE' }
AUTHOR : Robopac
VERSION : 0.0
// stored: AutoNumber false, IsOnlyStoredInLoadMemory false, IsWriteProtectedInAS false
   VAR RETAIN
      Program12 { S7_SetPoint := 'True'} : "DatiProgramma";
   END_VAR
BEGIN
   Program12.Wrapping := TRUE;
   Program12.TopLenght := 500;
   Program12.TopRelease := 0;
   Program12.TopDown := 0;
   Program12.Top := 4;
   Program12.PressurePTime := 0;
   Program12.LifterTime := 0;
   Program12.RevOverContrast := 1;
   Program12.RopeEndCycle := 16#02;
   Program12.Spare4 := 16#01;
   Program12.RopeTime := 1500;
   Program12.RevOverClamp := 1;
   Program12.FilmForceFinalRev := 10;
   Program12.FilmPrestretchFinalRev := 100;
   Program12.ArmSpeed := 100;
   Program12.CarriageDown4Top := 500;
   Program12.TopDownTime := 1500;
   Program12.LapsUnderTop := 0;
   Program12.Spare6 := 0;
   Program12.Spare7 := 0;
   Program12.Spare8 := 0;
   Program12.Spare9 := 0;
   Program12.Spare10 := 0;
   Program12.Spare11 := 0;
   Program12.Spare12 := 0;
   Program12.Overlap0_1 := 0;
   Program12.Height1 := 130;
   Program12.Landmark1 := FALSE;
   Program12.Lifter1 := FALSE;
   Program12.SpareBit1H1 := FALSE;
   Program12.Airblower1 := TRUE;
   Program12.NextStep1 := TRUE;
   Program12.PressureP1 := TRUE;
   Program12.SpareByte2H1 := 16#00;
   Program12.Revolution1 := 1;
   Program12.RopeUnit1_1 := 16#01;
   Program12.RopeUnit1_2 := 16#01;
   Program12.FilmForce1 := 5;
   Program12.FilmPrestretch1 := 200;
   Program12.Spare3H1 := 0;
   Program12.Spare49 := 0;
   Program12.Spare50 := 0;
   Program12.Spare51 := 0;
   Program12.Spare52 := 0;
   Program12.Spare53 := 0;
   Program12.Overlap1_2 := 0;
   Program12.Height2 := 50;
   Program12.Landmark2 := FALSE;
   Program12.Lifter2 := FALSE;
   Program12.SpareBit1H2 := FALSE;
   Program12.Airblower2 := TRUE;
   Program12.NextStep2 := TRUE;
   Program12.PressureP2 := TRUE;
   Program12.SpareByte2H2 := 16#00;
   Program12.Revolution2 := 1;
   Program12.RopeUnit2_1 := 16#01;
   Program12.RopeUnit2_2 := 16#01;
   Program12.FilmForce2 := 20;
   Program12.FilmPrestretch2 := 200;
   Program12.Spare3H2 := 0;
   Program12.Spare54 := 0;
   Program12.Spare55 := 0;
   Program12.Spare56 := 0;
   Program12.Spare57 := 0;
   Program12.Spare58 := 0;
   Program12.Overlap2_3 := 100;
   Program12.Height3 := -50;
   Program12.Landmark3 := TRUE;
   Program12.Lifter3 := FALSE;
   Program12.SpareBit1H3 := FALSE;
   Program12.Airblower3 := TRUE;
   Program12.NextStep3 := TRUE;
   Program12.PressureP3 := TRUE;
   Program12.SpareByte2H3 := 16#00;
   Program12.Revolution3 := 2;
   Program12.RopeUnit3_1 := 16#01;
   Program12.RopeUnit3_2 := 16#01;
   Program12.FilmForce3 := 30;
   Program12.FilmPrestretch3 := 200;
   Program12.Spare3H3 := 0;
   Program12.Spare59 := 0;
   Program12.Spare60 := 0;
   Program12.Spare61 := 380;
   Program12.Spare62 := 2800;
   Program12.Spare63 := 0;
   Program12.Overlap3_4 := 100;
   Program12.Height4 := 100;
   Program12.Landmark4 := FALSE;
   Program12.Lifter4 := FALSE;
   Program12.SpareBit1H4 := FALSE;
   Program12.Airblower4 := TRUE;
   Program12.NextStep4 := TRUE;
   Program12.PressureP4 := TRUE;
   Program12.SpareByte2H4 := 16#00;
   Program12.Revolution4 := 3;
   Program12.RopeUnit4_1 := 16#02;
   Program12.RopeUnit4_2 := 16#02;
   Program12.FilmForce4 := 30;
   Program12.FilmPrestretch4 := 200;
   Program12.Spare3H4 := 0;
   Program12.Spare64 := 0;
   Program12.Spare65 := 0;
   Program12.Spare66 := 0;
   Program12.Spare67 := 0;
   Program12.Spare68 := 0;
   Program12.Overlap4_5 := 0;
   Program12.Height5 := 50;
   Program12.Landmark5 := FALSE;
   Program12.Lifter5 := FALSE;
   Program12.SpareBit1H5 := FALSE;
   Program12.Airblower5 := TRUE;
   Program12.NextStep5 := FALSE;
   Program12.PressureP5 := FALSE;
   Program12.SpareByte2H5 := 16#00;
   Program12.Revolution5 := 1;
   Program12.RopeUnit5_1 := 16#01;
   Program12.RopeUnit5_2 := 16#01;
   Program12.FilmForce5 := 30;
   Program12.FilmPrestretch5 := 200;
   Program12.Spare3H5 := 0;
   Program12.Spare69 := 0;
   Program12.Spare70 := 0;
   Program12.Spare71 := 0;
   Program12.Spare72 := 0;
   Program12.Spare73 := 0;
   Program12.Overlap5_6 := 100;
   Program12.Height6 := 50;
   Program12.Landmark6 := FALSE;
   Program12.Lifter6 := FALSE;
   Program12.SpareBit1H6 := FALSE;
   Program12.Airblower6 := TRUE;
   Program12.NextStep6 := FALSE;
   Program12.PressureP6 := FALSE;
   Program12.SpareByte2H6 := 16#00;
   Program12.Revolution6 := 2;
   Program12.RopeUnit6_1 := 16#02;
   Program12.RopeUnit6_2 := 16#01;
   Program12.FilmForce6 := 20;
   Program12.FilmPrestretch6 := 200;
   Program12.Spare3H6 := 0;
   Program12.Spare74 := 0;
   Program12.Spare75 := 0;
   Program12.Spare76 := 0;
   Program12.Spare77 := 0;
   Program12.Spare78 := 0;
   Program12.Overlap6_7 := 0;
   Program12.Height7 := 0;
   Program12.Landmark7 := FALSE;
   Program12.Lifter7 := FALSE;
   Program12.SpareBit1H7 := FALSE;
   Program12.Airblower7 := FALSE;
   Program12.NextStep7 := TRUE;
   Program12.PressureP7 := FALSE;
   Program12.SpareByte2H7 := 16#00;
   Program12.Revolution7 := 1;
   Program12.RopeUnit7_1 := 16#01;
   Program12.RopeUnit7_2 := 16#01;
   Program12.FilmForce7 := 0;
   Program12.FilmPrestretch7 := 100;
   Program12.Spare3H7 := 0;
   Program12.Spare79 := 0;
   Program12.Spare80 := 0;
   Program12.Spare81 := 0;
   Program12.Spare82 := 0;
   Program12.Spare83 := 0;
   Program12.Overlap7_8 := 0;
   Program12.Height8 := 0;
   Program12.Landmark8 := FALSE;
   Program12.Lifter8 := FALSE;
   Program12.SpareBit1H8 := FALSE;
   Program12.Airblower8 := FALSE;
   Program12.NextStep8 := TRUE;
   Program12.PressureP8 := FALSE;
   Program12.SpareByte2H8 := 16#00;
   Program12.Revolution8 := 1;
   Program12.RopeUnit8_1 := 16#01;
   Program12.RopeUnit8_2 := 16#01;
   Program12.FilmForce8 := 0;
   Program12.FilmPrestretch8 := 100;
   Program12.Spare3H8 := 0;
   Program12.Spare84 := 0;
   Program12.Spare85 := 0;
   Program12.Spare86 := 0;
   Program12.Spare87 := 0;
   Program12.Spare88 := 0;
   Program12.Overlap8_9 := 0;
   Program12.Height9 := 0;
   Program12.Landmark9 := FALSE;
   Program12.Lifter9 := FALSE;
   Program12.SpareBit1H9 := FALSE;
   Program12.Airblower9 := FALSE;
   Program12.NextStep9 := TRUE;
   Program12.PressureP9 := FALSE;
   Program12.SpareByte2H9 := 16#00;
   Program12.Revolution9 := 1;
   Program12.RopeUnit9_1 := 16#01;
   Program12.RopeUnit9_2 := 16#01;
   Program12.FilmForce9 := 0;
   Program12.FilmPrestretch9 := 100;
   Program12.Spare3H9 := 0;
   Program12.Spare89 := 0;
   Program12.Spare90 := 0;
   Program12.Spare91 := 0;
   Program12.Spare92 := 0;
   Program12.Spare93 := 0;
   Program12.Overlap9_10 := 0;
   Program12.Height10 := 0;
   Program12.Landmark10 := FALSE;
   Program12.Lifter10 := FALSE;
   Program12.SpareBit1H10 := FALSE;
   Program12.Airblower10 := FALSE;
   Program12.NextStep10 := FALSE;
   Program12.PressureP10 := FALSE;
   Program12.SpareByte2H10 := 16#00;
   Program12.Revolution10 := 1;
   Program12.RopeUnit10_1 := 16#01;
   Program12.RopeUnit10_2 := 16#01;
   Program12.FilmForce10 := 0;
   Program12.FilmPrestretch10 := 100;
   Program12.Spare3H10 := 0;
   Program12.Spare94 := 0;
   Program12.Spare95 := 0;
   Program12.Spare96 := 0;
   Program12.Spare97 := 0;
   Program12.Spare98 := 0;
   Program12.Overlap10_11 := 0;
   Program12.Height11 := 0;
   Program12.Landmark11 := FALSE;
   Program12.Lifter11 := FALSE;
   Program12.SpareBit1H11 := FALSE;
   Program12.Airblower11 := FALSE;
   Program12.NextStep11 := TRUE;
   Program12.PressureP11 := FALSE;
   Program12.SpareByte2H11 := 16#00;
   Program12.Revolution11 := 1;
   Program12.RopeUnit11_1 := 16#01;
   Program12.RopeUnit11_2 := 16#01;
   Program12.FilmForce11 := 0;
   Program12.FilmPrestretch11 := 100;
   Program12.Spare3H11 := 0;
   Program12.Spare99 := 0;
   Program12.Spare100 := 0;
   Program12.Spare101 := 0;
   Program12.Spare102 := 0;
   Program12.Spare103 := 0;
   Program12.Overlap11_12 := 0;
   Program12.Height12 := 0;
   Program12.Landmark12 := FALSE;
   Program12.Lifter12 := FALSE;
   Program12.SpareBit1H12 := FALSE;
   Program12.Airblower12 := FALSE;
   Program12.NextStep12 := FALSE;
   Program12.PressureP12 := FALSE;
   Program12.SpareByte2H12 := 16#00;
   Program12.Revolution12 := 1;
   Program12.RopeUnit12_1 := 16#01;
   Program12.RopeUnit12_2 := 16#01;
   Program12.FilmForce12 := 0;
   Program12.FilmPrestretch12 := 100;
   Program12.Spare3H12 := 0;
   Program12.Spare104 := 0;
   Program12.Spare105 := 0;
   Program12.Spare106 := 0;
   Program12.Spare107 := 0;
   Program12.Spare108 := 0;
END_DATA_BLOCK

DATA_BLOCK "DB239_Program11"   // DB239
{ S7_Optimized_Access := 'FALSE' }
AUTHOR : Robopac
VERSION : 0.0
// stored: AutoNumber false, IsOnlyStoredInLoadMemory false, IsWriteProtectedInAS false
   VAR RETAIN
      Program11 { S7_SetPoint := 'True'} : "DatiProgramma";
   END_VAR
BEGIN
   Program11.Wrapping := TRUE;
   Program11.TopLenght := 500;
   Program11.TopRelease := 0;
   Program11.TopDown := 0;
   Program11.Top := 4;
   Program11.PressurePTime := 0;
   Program11.LifterTime := 0;
   Program11.RevOverContrast := 1;
   Program11.RopeEndCycle := 16#02;
   Program11.Spare4 := 16#01;
   Program11.RopeTime := 1500;
   Program11.RevOverClamp := 1;
   Program11.FilmForceFinalRev := 10;
   Program11.FilmPrestretchFinalRev := 100;
   Program11.ArmSpeed := 100;
   Program11.CarriageDown4Top := 500;
   Program11.TopDownTime := 1500;
   Program11.LapsUnderTop := 0;
   Program11.Spare6 := 0;
   Program11.Spare7 := 0;
   Program11.Spare8 := 0;
   Program11.Spare9 := 0;
   Program11.Spare10 := 0;
   Program11.Spare11 := 0;
   Program11.Spare12 := 0;
   Program11.Overlap0_1 := 0;
   Program11.Height1 := 130;
   Program11.Landmark1 := FALSE;
   Program11.Lifter1 := FALSE;
   Program11.SpareBit1H1 := FALSE;
   Program11.Airblower1 := TRUE;
   Program11.NextStep1 := TRUE;
   Program11.PressureP1 := TRUE;
   Program11.SpareByte2H1 := 16#00;
   Program11.Revolution1 := 1;
   Program11.RopeUnit1_1 := 16#01;
   Program11.RopeUnit1_2 := 16#01;
   Program11.FilmForce1 := 5;
   Program11.FilmPrestretch1 := 200;
   Program11.Spare3H1 := 0;
   Program11.Spare49 := 0;
   Program11.Spare50 := 0;
   Program11.Spare51 := 0;
   Program11.Spare52 := 0;
   Program11.Spare53 := 0;
   Program11.Overlap1_2 := 0;
   Program11.Height2 := 50;
   Program11.Landmark2 := FALSE;
   Program11.Lifter2 := FALSE;
   Program11.SpareBit1H2 := FALSE;
   Program11.Airblower2 := TRUE;
   Program11.NextStep2 := TRUE;
   Program11.PressureP2 := TRUE;
   Program11.SpareByte2H2 := 16#00;
   Program11.Revolution2 := 1;
   Program11.RopeUnit2_1 := 16#01;
   Program11.RopeUnit2_2 := 16#01;
   Program11.FilmForce2 := 20;
   Program11.FilmPrestretch2 := 200;
   Program11.Spare3H2 := 0;
   Program11.Spare54 := 0;
   Program11.Spare55 := 0;
   Program11.Spare56 := 0;
   Program11.Spare57 := 0;
   Program11.Spare58 := 0;
   Program11.Overlap2_3 := 100;
   Program11.Height3 := -50;
   Program11.Landmark3 := TRUE;
   Program11.Lifter3 := FALSE;
   Program11.SpareBit1H3 := FALSE;
   Program11.Airblower3 := TRUE;
   Program11.NextStep3 := TRUE;
   Program11.PressureP3 := TRUE;
   Program11.SpareByte2H3 := 16#00;
   Program11.Revolution3 := 2;
   Program11.RopeUnit3_1 := 16#01;
   Program11.RopeUnit3_2 := 16#01;
   Program11.FilmForce3 := 30;
   Program11.FilmPrestretch3 := 200;
   Program11.Spare3H3 := 0;
   Program11.Spare59 := 0;
   Program11.Spare60 := 0;
   Program11.Spare61 := 380;
   Program11.Spare62 := 2800;
   Program11.Spare63 := 0;
   Program11.Overlap3_4 := 100;
   Program11.Height4 := 100;
   Program11.Landmark4 := FALSE;
   Program11.Lifter4 := FALSE;
   Program11.SpareBit1H4 := FALSE;
   Program11.Airblower4 := TRUE;
   Program11.NextStep4 := TRUE;
   Program11.PressureP4 := TRUE;
   Program11.SpareByte2H4 := 16#00;
   Program11.Revolution4 := 3;
   Program11.RopeUnit4_1 := 16#02;
   Program11.RopeUnit4_2 := 16#02;
   Program11.FilmForce4 := 30;
   Program11.FilmPrestretch4 := 200;
   Program11.Spare3H4 := 0;
   Program11.Spare64 := 0;
   Program11.Spare65 := 0;
   Program11.Spare66 := 0;
   Program11.Spare67 := 0;
   Program11.Spare68 := 0;
   Program11.Overlap4_5 := 0;
   Program11.Height5 := 50;
   Program11.Landmark5 := FALSE;
   Program11.Lifter5 := FALSE;
   Program11.SpareBit1H5 := FALSE;
   Program11.Airblower5 := TRUE;
   Program11.NextStep5 := FALSE;
   Program11.PressureP5 := FALSE;
   Program11.SpareByte2H5 := 16#00;
   Program11.Revolution5 := 1;
   Program11.RopeUnit5_1 := 16#01;
   Program11.RopeUnit5_2 := 16#01;
   Program11.FilmForce5 := 30;
   Program11.FilmPrestretch5 := 200;
   Program11.Spare3H5 := 0;
   Program11.Spare69 := 0;
   Program11.Spare70 := 0;
   Program11.Spare71 := 0;
   Program11.Spare72 := 0;
   Program11.Spare73 := 0;
   Program11.Overlap5_6 := 100;
   Program11.Height6 := 50;
   Program11.Landmark6 := FALSE;
   Program11.Lifter6 := FALSE;
   Program11.SpareBit1H6 := FALSE;
   Program11.Airblower6 := TRUE;
   Program11.NextStep6 := FALSE;
   Program11.PressureP6 := FALSE;
   Program11.SpareByte2H6 := 16#00;
   Program11.Revolution6 := 2;
   Program11.RopeUnit6_1 := 16#02;
   Program11.RopeUnit6_2 := 16#01;
   Program11.FilmForce6 := 20;
   Program11.FilmPrestretch6 := 200;
   Program11.Spare3H6 := 0;
   Program11.Spare74 := 0;
   Program11.Spare75 := 0;
   Program11.Spare76 := 0;
   Program11.Spare77 := 0;
   Program11.Spare78 := 0;
   Program11.Overlap6_7 := 0;
   Program11.Height7 := 0;
   Program11.Landmark7 := FALSE;
   Program11.Lifter7 := FALSE;
   Program11.SpareBit1H7 := FALSE;
   Program11.Airblower7 := FALSE;
   Program11.NextStep7 := TRUE;
   Program11.PressureP7 := FALSE;
   Program11.SpareByte2H7 := 16#00;
   Program11.Revolution7 := 1;
   Program11.RopeUnit7_1 := 16#01;
   Program11.RopeUnit7_2 := 16#01;
   Program11.FilmForce7 := 0;
   Program11.FilmPrestretch7 := 100;
   Program11.Spare3H7 := 0;
   Program11.Spare79 := 0;
   Program11.Spare80 := 0;
   Program11.Spare81 := 0;
   Program11.Spare82 := 0;
   Program11.Spare83 := 0;
   Program11.Overlap7_8 := 0;
   Program11.Height8 := 0;
   Program11.Landmark8 := FALSE;
   Program11.Lifter8 := FALSE;
   Program11.SpareBit1H8 := FALSE;
   Program11.Airblower8 := FALSE;
   Program11.NextStep8 := TRUE;
   Program11.PressureP8 := FALSE;
   Program11.SpareByte2H8 := 16#00;
   Program11.Revolution8 := 1;
   Program11.RopeUnit8_1 := 16#01;
   Program11.RopeUnit8_2 := 16#01;
   Program11.FilmForce8 := 0;
   Program11.FilmPrestretch8 := 100;
   Program11.Spare3H8 := 0;
   Program11.Spare84 := 0;
   Program11.Spare85 := 0;
   Program11.Spare86 := 0;
   Program11.Spare87 := 0;
   Program11.Spare88 := 0;
   Program11.Overlap8_9 := 0;
   Program11.Height9 := 0;
   Program11.Landmark9 := FALSE;
   Program11.Lifter9 := FALSE;
   Program11.SpareBit1H9 := FALSE;
   Program11.Airblower9 := FALSE;
   Program11.NextStep9 := TRUE;
   Program11.PressureP9 := FALSE;
   Program11.SpareByte2H9 := 16#00;
   Program11.Revolution9 := 1;
   Program11.RopeUnit9_1 := 16#01;
   Program11.RopeUnit9_2 := 16#01;
   Program11.FilmForce9 := 0;
   Program11.FilmPrestretch9 := 100;
   Program11.Spare3H9 := 0;
   Program11.Spare89 := 0;
   Program11.Spare90 := 0;
   Program11.Spare91 := 0;
   Program11.Spare92 := 0;
   Program11.Spare93 := 0;
   Program11.Overlap9_10 := 0;
   Program11.Height10 := 0;
   Program11.Landmark10 := FALSE;
   Program11.Lifter10 := FALSE;
   Program11.SpareBit1H10 := FALSE;
   Program11.Airblower10 := FALSE;
   Program11.NextStep10 := FALSE;
   Program11.PressureP10 := FALSE;
   Program11.SpareByte2H10 := 16#00;
   Program11.Revolution10 := 1;
   Program11.RopeUnit10_1 := 16#01;
   Program11.RopeUnit10_2 := 16#01;
   Program11.FilmForce10 := 0;
   Program11.FilmPrestretch10 := 100;
   Program11.Spare3H10 := 0;
   Program11.Spare94 := 0;
   Program11.Spare95 := 0;
   Program11.Spare96 := 0;
   Program11.Spare97 := 0;
   Program11.Spare98 := 0;
   Program11.Overlap10_11 := 0;
   Program11.Height11 := 0;
   Program11.Landmark11 := FALSE;
   Program11.Lifter11 := FALSE;
   Program11.SpareBit1H11 := FALSE;
   Program11.Airblower11 := FALSE;
   Program11.NextStep11 := TRUE;
   Program11.PressureP11 := FALSE;
   Program11.SpareByte2H11 := 16#00;
   Program11.Revolution11 := 1;
   Program11.RopeUnit11_1 := 16#01;
   Program11.RopeUnit11_2 := 16#01;
   Program11.FilmForce11 := 0;
   Program11.FilmPrestretch11 := 100;
   Program11.Spare3H11 := 0;
   Program11.Spare99 := 0;
   Program11.Spare100 := 0;
   Program11.Spare101 := 0;
   Program11.Spare102 := 0;
   Program11.Spare103 := 0;
   Program11.Overlap11_12 := 0;
   Program11.Height12 := 0;
   Program11.Landmark12 := FALSE;
   Program11.Lifter12 := FALSE;
   Program11.SpareBit1H12 := FALSE;
   Program11.Airblower12 := FALSE;
   Program11.NextStep12 := FALSE;
   Program11.PressureP12 := FALSE;
   Program11.SpareByte2H12 := 16#00;
   Program11.Revolution12 := 1;
   Program11.RopeUnit12_1 := 16#01;
   Program11.RopeUnit12_2 := 16#01;
   Program11.FilmForce12 := 0;
   Program11.FilmPrestretch12 := 100;
   Program11.Spare3H12 := 0;
   Program11.Spare104 := 0;
   Program11.Spare105 := 0;
   Program11.Spare106 := 0;
   Program11.Spare107 := 0;
   Program11.Spare108 := 0;
END_DATA_BLOCK

DATA_BLOCK "DB241_Program9"   // DB241
{ S7_Optimized_Access := 'FALSE' }
AUTHOR : Robopac
VERSION : 0.0
// stored: AutoNumber false, IsOnlyStoredInLoadMemory false, IsWriteProtectedInAS false
   VAR RETAIN
      Program9 { S7_SetPoint := 'True'} : "DatiProgramma";
   END_VAR
BEGIN
   Program9.Wrapping := TRUE;
   Program9.TopLenght := 500;
   Program9.TopRelease := 0;
   Program9.TopDown := 0;
   Program9.Top := 4;
   Program9.PressurePTime := 0;
   Program9.LifterTime := 0;
   Program9.RevOverContrast := 1;
   Program9.RopeEndCycle := 16#02;
   Program9.Spare4 := 16#01;
   Program9.RopeTime := 1500;
   Program9.RevOverClamp := 1;
   Program9.FilmForceFinalRev := 10;
   Program9.FilmPrestretchFinalRev := 100;
   Program9.ArmSpeed := 100;
   Program9.CarriageDown4Top := 500;
   Program9.TopDownTime := 1500;
   Program9.LapsUnderTop := 0;
   Program9.Spare6 := 0;
   Program9.Spare7 := 0;
   Program9.Spare8 := 0;
   Program9.Spare9 := 0;
   Program9.Spare10 := 0;
   Program9.Spare11 := 0;
   Program9.Spare12 := 0;
   Program9.Overlap0_1 := 0;
   Program9.Height1 := 130;
   Program9.Landmark1 := FALSE;
   Program9.Lifter1 := FALSE;
   Program9.SpareBit1H1 := FALSE;
   Program9.Airblower1 := TRUE;
   Program9.NextStep1 := TRUE;
   Program9.PressureP1 := TRUE;
   Program9.SpareByte2H1 := 16#00;
   Program9.Revolution1 := 1;
   Program9.RopeUnit1_1 := 16#01;
   Program9.RopeUnit1_2 := 16#01;
   Program9.FilmForce1 := 5;
   Program9.FilmPrestretch1 := 200;
   Program9.Spare3H1 := 0;
   Program9.Spare49 := 0;
   Program9.Spare50 := 0;
   Program9.Spare51 := 0;
   Program9.Spare52 := 0;
   Program9.Spare53 := 0;
   Program9.Overlap1_2 := 0;
   Program9.Height2 := 50;
   Program9.Landmark2 := FALSE;
   Program9.Lifter2 := FALSE;
   Program9.SpareBit1H2 := FALSE;
   Program9.Airblower2 := TRUE;
   Program9.NextStep2 := TRUE;
   Program9.PressureP2 := TRUE;
   Program9.SpareByte2H2 := 16#00;
   Program9.Revolution2 := 1;
   Program9.RopeUnit2_1 := 16#01;
   Program9.RopeUnit2_2 := 16#01;
   Program9.FilmForce2 := 20;
   Program9.FilmPrestretch2 := 200;
   Program9.Spare3H2 := 0;
   Program9.Spare54 := 0;
   Program9.Spare55 := 0;
   Program9.Spare56 := 0;
   Program9.Spare57 := 0;
   Program9.Spare58 := 0;
   Program9.Overlap2_3 := 100;
   Program9.Height3 := -50;
   Program9.Landmark3 := TRUE;
   Program9.Lifter3 := FALSE;
   Program9.SpareBit1H3 := FALSE;
   Program9.Airblower3 := TRUE;
   Program9.NextStep3 := TRUE;
   Program9.PressureP3 := TRUE;
   Program9.SpareByte2H3 := 16#00;
   Program9.Revolution3 := 2;
   Program9.RopeUnit3_1 := 16#01;
   Program9.RopeUnit3_2 := 16#01;
   Program9.FilmForce3 := 30;
   Program9.FilmPrestretch3 := 200;
   Program9.Spare3H3 := 0;
   Program9.Spare59 := 0;
   Program9.Spare60 := 0;
   Program9.Spare61 := 380;
   Program9.Spare62 := 2800;
   Program9.Spare63 := 0;
   Program9.Overlap3_4 := 100;
   Program9.Height4 := 100;
   Program9.Landmark4 := FALSE;
   Program9.Lifter4 := FALSE;
   Program9.SpareBit1H4 := FALSE;
   Program9.Airblower4 := TRUE;
   Program9.NextStep4 := TRUE;
   Program9.PressureP4 := TRUE;
   Program9.SpareByte2H4 := 16#00;
   Program9.Revolution4 := 3;
   Program9.RopeUnit4_1 := 16#02;
   Program9.RopeUnit4_2 := 16#02;
   Program9.FilmForce4 := 30;
   Program9.FilmPrestretch4 := 200;
   Program9.Spare3H4 := 0;
   Program9.Spare64 := 0;
   Program9.Spare65 := 0;
   Program9.Spare66 := 0;
   Program9.Spare67 := 0;
   Program9.Spare68 := 0;
   Program9.Overlap4_5 := 0;
   Program9.Height5 := 50;
   Program9.Landmark5 := FALSE;
   Program9.Lifter5 := FALSE;
   Program9.SpareBit1H5 := FALSE;
   Program9.Airblower5 := TRUE;
   Program9.NextStep5 := FALSE;
   Program9.PressureP5 := FALSE;
   Program9.SpareByte2H5 := 16#00;
   Program9.Revolution5 := 1;
   Program9.RopeUnit5_1 := 16#01;
   Program9.RopeUnit5_2 := 16#01;
   Program9.FilmForce5 := 30;
   Program9.FilmPrestretch5 := 200;
   Program9.Spare3H5 := 0;
   Program9.Spare69 := 0;
   Program9.Spare70 := 0;
   Program9.Spare71 := 0;
   Program9.Spare72 := 0;
   Program9.Spare73 := 0;
   Program9.Overlap5_6 := 100;
   Program9.Height6 := 50;
   Program9.Landmark6 := FALSE;
   Program9.Lifter6 := FALSE;
   Program9.SpareBit1H6 := FALSE;
   Program9.Airblower6 := TRUE;
   Program9.NextStep6 := FALSE;
   Program9.PressureP6 := FALSE;
   Program9.SpareByte2H6 := 16#00;
   Program9.Revolution6 := 2;
   Program9.RopeUnit6_1 := 16#02;
   Program9.RopeUnit6_2 := 16#01;
   Program9.FilmForce6 := 20;
   Program9.FilmPrestretch6 := 200;
   Program9.Spare3H6 := 0;
   Program9.Spare74 := 0;
   Program9.Spare75 := 0;
   Program9.Spare76 := 0;
   Program9.Spare77 := 0;
   Program9.Spare78 := 0;
   Program9.Overlap6_7 := 0;
   Program9.Height7 := 0;
   Program9.Landmark7 := FALSE;
   Program9.Lifter7 := FALSE;
   Program9.SpareBit1H7 := FALSE;
   Program9.Airblower7 := FALSE;
   Program9.NextStep7 := TRUE;
   Program9.PressureP7 := FALSE;
   Program9.SpareByte2H7 := 16#00;
   Program9.Revolution7 := 1;
   Program9.RopeUnit7_1 := 16#01;
   Program9.RopeUnit7_2 := 16#01;
   Program9.FilmForce7 := 0;
   Program9.FilmPrestretch7 := 100;
   Program9.Spare3H7 := 0;
   Program9.Spare79 := 0;
   Program9.Spare80 := 0;
   Program9.Spare81 := 0;
   Program9.Spare82 := 0;
   Program9.Spare83 := 0;
   Program9.Overlap7_8 := 0;
   Program9.Height8 := 0;
   Program9.Landmark8 := FALSE;
   Program9.Lifter8 := FALSE;
   Program9.SpareBit1H8 := FALSE;
   Program9.Airblower8 := FALSE;
   Program9.NextStep8 := TRUE;
   Program9.PressureP8 := FALSE;
   Program9.SpareByte2H8 := 16#00;
   Program9.Revolution8 := 1;
   Program9.RopeUnit8_1 := 16#01;
   Program9.RopeUnit8_2 := 16#01;
   Program9.FilmForce8 := 0;
   Program9.FilmPrestretch8 := 100;
   Program9.Spare3H8 := 0;
   Program9.Spare84 := 0;
   Program9.Spare85 := 0;
   Program9.Spare86 := 0;
   Program9.Spare87 := 0;
   Program9.Spare88 := 0;
   Program9.Overlap8_9 := 0;
   Program9.Height9 := 0;
   Program9.Landmark9 := FALSE;
   Program9.Lifter9 := FALSE;
   Program9.SpareBit1H9 := FALSE;
   Program9.Airblower9 := FALSE;
   Program9.NextStep9 := TRUE;
   Program9.PressureP9 := FALSE;
   Program9.SpareByte2H9 := 16#00;
   Program9.Revolution9 := 1;
   Program9.RopeUnit9_1 := 16#01;
   Program9.RopeUnit9_2 := 16#01;
   Program9.FilmForce9 := 0;
   Program9.FilmPrestretch9 := 100;
   Program9.Spare3H9 := 0;
   Program9.Spare89 := 0;
   Program9.Spare90 := 0;
   Program9.Spare91 := 0;
   Program9.Spare92 := 0;
   Program9.Spare93 := 0;
   Program9.Overlap9_10 := 0;
   Program9.Height10 := 0;
   Program9.Landmark10 := FALSE;
   Program9.Lifter10 := FALSE;
   Program9.SpareBit1H10 := FALSE;
   Program9.Airblower10 := FALSE;
   Program9.NextStep10 := FALSE;
   Program9.PressureP10 := FALSE;
   Program9.SpareByte2H10 := 16#00;
   Program9.Revolution10 := 1;
   Program9.RopeUnit10_1 := 16#01;
   Program9.RopeUnit10_2 := 16#01;
   Program9.FilmForce10 := 0;
   Program9.FilmPrestretch10 := 100;
   Program9.Spare3H10 := 0;
   Program9.Spare94 := 0;
   Program9.Spare95 := 0;
   Program9.Spare96 := 0;
   Program9.Spare97 := 0;
   Program9.Spare98 := 0;
   Program9.Overlap10_11 := 0;
   Program9.Height11 := 0;
   Program9.Landmark11 := FALSE;
   Program9.Lifter11 := FALSE;
   Program9.SpareBit1H11 := FALSE;
   Program9.Airblower11 := FALSE;
   Program9.NextStep11 := TRUE;
   Program9.PressureP11 := FALSE;
   Program9.SpareByte2H11 := 16#00;
   Program9.Revolution11 := 1;
   Program9.RopeUnit11_1 := 16#01;
   Program9.RopeUnit11_2 := 16#01;
   Program9.FilmForce11 := 0;
   Program9.FilmPrestretch11 := 100;
   Program9.Spare3H11 := 0;
   Program9.Spare99 := 0;
   Program9.Spare100 := 0;
   Program9.Spare101 := 0;
   Program9.Spare102 := 0;
   Program9.Spare103 := 0;
   Program9.Overlap11_12 := 0;
   Program9.Height12 := 0;
   Program9.Landmark12 := FALSE;
   Program9.Lifter12 := FALSE;
   Program9.SpareBit1H12 := FALSE;
   Program9.Airblower12 := FALSE;
   Program9.NextStep12 := FALSE;
   Program9.PressureP12 := FALSE;
   Program9.SpareByte2H12 := 16#00;
   Program9.Revolution12 := 1;
   Program9.RopeUnit12_1 := 16#01;
   Program9.RopeUnit12_2 := 16#01;
   Program9.FilmForce12 := 0;
   Program9.FilmPrestretch12 := 100;
   Program9.Spare3H12 := 0;
   Program9.Spare104 := 0;
   Program9.Spare105 := 0;
   Program9.Spare106 := 0;
   Program9.Spare107 := 0;
   Program9.Spare108 := 0;
END_DATA_BLOCK

